(* IEC 61131-3 sources: ml2plc/benchmarks/st (part 14) *)

VAR
    (* Merged variables from all regions *)
    buffer_0 : ARRAY[0..63] OF REAL;
    buffer_1 : ARRAY[0..63] OF REAL;
    c_state_0 : ARRAY[0..63] OF REAL;
    c_state_3 : ARRAY[0..63] OF REAL;
    f_gate_0 : ARRAY[0..63] OF REAL;
    f_gate_3 : ARRAY[0..63] OF REAL;
    g_gate_0 : ARRAY[0..63] OF REAL;
    g_gate_3 : ARRAY[0..63] OF REAL;
    h_state_0 : ARRAY[0..63] OF REAL;
    h_state_3 : ARRAY[0..63] OF REAL;
    i_gate_0 : ARRAY[0..63] OF REAL;
    i_gate_3 : ARRAY[0..63] OF REAL;
    o_gate_0 : ARRAY[0..63] OF REAL;
    o_gate_3 : ARRAY[0..63] OF REAL;

    (* Temporary computation variables *)
    i : DINT;
    j : DINT;
    t : DINT;
    sum : REAL;
    (* Computation helpers *)
    max_val : REAL;
    exp_val : REAL;
    exp_sum : REAL;
    (* Spatial loop variables *)
    oc : DINT;
    oh : DINT;
    ow : DINT;
    ic : DINT;
    kh : DINT;
    kw : DINT;
    ih : DINT;
    iw : DINT;
    (* Transpose loop variables *)
    t2_d0 : DINT;
    t2_d1 : DINT;
    t2_d2 : DINT;
END_VAR

(* Forward pass execution *)

(* Region: r0 [ACYCLIC] *)
(* Acyclic Region r0 *)
(* Layer 0: LSTM (hidden_size=64, input_size=1, seq_len=1) *)
(* Generating output: Y *)

(* Initialize states to zero *)
FOR j := 0 TO 63 DO
    h_state_0[j] := 0.0;
    c_state_0[j] := 0.0;
END_FOR;

(* Process 1 timesteps *)
FOR t := 0 TO 0 DO

    (* Input Gate *)
    FOR j := 0 TO 63 DO
        sum := 0.0;
        FOR i := 0 TO 0 DO
            sum := sum + input_data * weights_0_i[j * 1 + i] ;
        END_FOR;
        FOR i := 0 TO 63 DO
            sum := sum + h_state_0[i] * recurrent_0_i[j * 64 + i] ;
        END_FOR;
    sum := sum + bias_0_i[j];
    i_gate_0[j] := 1.0 / (1.0 + EXP(-sum));
    END_FOR;

    (* Forget Gate *)
    FOR j := 0 TO 63 DO
        sum := 0.0;
        FOR i := 0 TO 0 DO
            sum := sum + input_data * weights_0_f[j * 1 + i] ;
        END_FOR;
        FOR i := 0 TO 63 DO
            sum := sum + h_state_0[i] * recurrent_0_f[j * 64 + i] ;
        END_FOR;
    sum := sum + bias_0_f[j];
    f_gate_0[j] := 1.0 / (1.0 + EXP(-sum));
    END_FOR;

    (* Cell Gate *)
    FOR j := 0 TO 63 DO
        sum := 0.0;
        FOR i := 0 TO 0 DO
            sum := sum + input_data * weights_0_g[j * 1 + i] ;
        END_FOR;
        FOR i := 0 TO 63 DO
            sum := sum + h_state_0[i] * recurrent_0_g[j * 64 + i] ;
        END_FOR;
    sum := sum + bias_0_g[j];
    exp_val := EXP(2.0 * sum);
    g_gate_0[j] := (exp_val - 1.0) / (exp_val + 1.0);
    END_FOR;

    (* Output Gate *)
    FOR j := 0 TO 63 DO
        sum := 0.0;
        FOR i := 0 TO 0 DO
            sum := sum + input_data * weights_0_o[j * 1 + i] ;
        END_FOR;
        FOR i := 0 TO 63 DO
            sum := sum + h_state_0[i] * recurrent_0_o[j * 64 + i] ;
        END_FOR;
    sum := sum + bias_0_o[j];
    o_gate_0[j] := 1.0 / (1.0 + EXP(-sum));
    END_FOR;

    (* Cell state: c_t = f_t * c_{t-1} + i_t * g_t *)
    FOR j := 0 TO 63 DO
        c_state_0[j] := f_gate_0[j] * c_state_0[j] + i_gate_0[j] * g_gate_0[j];
    END_FOR;

    (* Hidden state: h_t = o_t * tanh(c_t) *)
    FOR j := 0 TO 63 DO
        exp_val := EXP(2.0 * c_state_0[j]);
        h_state_0[j] := o_gate_0[j] * ((exp_val - 1.0) / (exp_val + 1.0));
    END_FOR;

    (* Y output: Full sequence *)
    FOR j := 0 TO 63 DO
        buffer_0[t * 64 + j] := h_state_0[j];
    END_FOR;
END_FOR;

(* Layer 1: Squeeze *)
FOR i := 0 TO 63 DO
    buffer_1[i] := buffer_0[i];
END_FOR;

(* Layer 2: Transpose perm=(1, 0, 2)  (1, 1, 64) -> (1, 1, 64) *)
FOR t2_d0 := 0 TO 0 DO
    FOR t2_d1 := 0 TO 0 DO
        FOR t2_d2 := 0 TO 63 DO
            buffer_0[t2_d0 * 64 + t2_d1 * 64 + t2_d2] := buffer_1[t2_d1 * 64 + t2_d0 * 64 + t2_d2];
        END_FOR;
    END_FOR;
END_FOR;

(* Layer 3: LSTM (hidden_size=64, input_size=64, seq_len=1) *)
(* Generating output: Y *)

(* Initialize states to zero *)
FOR j := 0 TO 63 DO
    h_state_3[j] := 0.0;
    c_state_3[j] := 0.0;
END_FOR;

(* Process 1 timesteps *)
FOR t := 0 TO 0 DO

    (* Input Gate *)
    FOR j := 0 TO 63 DO
        sum := 0.0;
        FOR i := 0 TO 63 DO
            sum := sum + buffer_0[t * 64 + i] * weights_3_i[j * 64 + i] ;
        END_FOR;
        FOR i := 0 TO 63 DO
            sum := sum + h_state_3[i] * recurrent_3_i[j * 64 + i] ;
        END_FOR;
    sum := sum + bias_3_i[j];
    i_gate_3[j] := 1.0 / (1.0 + EXP(-sum));
    END_FOR;

    (* Forget Gate *)
    FOR j := 0 TO 63 DO
        sum := 0.0;
        FOR i := 0 TO 63 DO
            sum := sum + buffer_0[t * 64 + i] * weights_3_f[j * 64 + i] ;
        END_FOR;
        FOR i := 0 TO 63 DO
            sum := sum + h_state_3[i] * recurrent_3_f[j * 64 + i] ;
        END_FOR;
    sum := sum + bias_3_f[j];
    f_gate_3[j] := 1.0 / (1.0 + EXP(-sum));
    END_FOR;

    (* Cell Gate *)
    FOR j := 0 TO 63 DO
        sum := 0.0;
        FOR i := 0 TO 63 DO
            sum := sum + buffer_0[t * 64 + i] * weights_3_g[j * 64 + i] ;
        END_FOR;
        FOR i := 0 TO 63 DO
            sum := sum + h_state_3[i] * recurrent_3_g[j * 64 + i] ;
        END_FOR;
    sum := sum + bias_3_g[j];
    exp_val := EXP(2.0 * sum);
    g_gate_3[j] := (exp_val - 1.0) / (exp_val + 1.0);
    END_FOR;

    (* Output Gate *)
    FOR j := 0 TO 63 DO
        sum := 0.0;
        FOR i := 0 TO 63 DO
            sum := sum + buffer_0[t * 64 + i] * weights_3_o[j * 64 + i] ;
        END_FOR;
        FOR i := 0 TO 63 DO
            sum := sum + h_state_3[i] * recurrent_3_o[j * 64 + i] ;
        END_FOR;
    sum := sum + bias_3_o[j];
    o_gate_3[j] := 1.0 / (1.0 + EXP(-sum));
    END_FOR;

    (* Cell state: c_t = f_t * c_{t-1} + i_t * g_t *)
    FOR j := 0 TO 63 DO
        c_state_3[j] := f_gate_3[j] * c_state_3[j] + i_gate_3[j] * g_gate_3[j];
    END_FOR;

    (* Hidden state: h_t = o_t * tanh(c_t) *)
    FOR j := 0 TO 63 DO
        exp_val := EXP(2.0 * c_state_3[j]);
        h_state_3[j] := o_gate_3[j] * ((exp_val - 1.0) / (exp_val + 1.0));
    END_FOR;

    (* Y output: Full sequence *)
    FOR j := 0 TO 63 DO
        buffer_1[t * 64 + j] := h_state_3[j];
    END_FOR;
END_FOR;

(* Layer 4: Squeeze *)
FOR i := 0 TO 63 DO
    buffer_0[i] := buffer_1[i];
END_FOR;

(* Layer 5: Slice starts=[0] ends=[1] axes=[0] steps=[1] *)
FOR i := 0 TO 63 DO
    buffer_1[i] := buffer_0[i];
END_FOR;

(* Layer 6: Squeeze *)
FOR i := 0 TO 63 DO
    buffer_0[i] := buffer_1[i];
END_FOR;

(* Layer 7: Fused Linear + SOFTMAX *)
FOR j := 0 TO 2 DO
    sum := 0.0;
    FOR i := 0 TO 63 DO
        sum := sum + buffer_0[i] * weights_7[i * 3 + j];
    END_FOR;
output_data[j] := sum + bias_7[j];
END_FOR;

(* Softmax: find max *)
max_val := output_data[0];
FOR i := 1 TO 2 DO
    IF output_data[i] > max_val THEN
        max_val := output_data[i];
    END_IF;
END_FOR;

(* Softmax: compute exponentials and sum *)
exp_sum := 0.0;
FOR i := 0 TO 2 DO
    output_data[i] := EXP(output_data[i] - max_val);
    exp_sum := exp_sum + output_data[i];
END_FOR;

(* Softmax: normalize *)
FOR i := 0 TO 2 DO
    output_data[i] := output_data[i] / exp_sum;
END_FOR;

END_FUNCTION_BLOCK

(* ---- MLP1.st ---- *)
FUNCTION_BLOCK MLP1_FB

    (* Model Inputs/Outputs *)
VAR_INPUT
    input_data : REAL;
END_VAR

VAR_OUTPUT
    output_data : ARRAY[0..2] OF REAL;
END_VAR

VAR CONSTANT
    weights_0 : ARRAY[0..7] OF REAL := [-0.39633444, -0.548940063, -0.0548924804, 2.65775609, -0.186861873, 1.99443269, -0.4275029, 2.42555642];
    bias_0 : ARRAY[0..7] OF REAL := [0, 0, 0, -0.386175603, 1.51318884, -0.335069925, 0, -0.41231662];

    weights_1 : ARRAY[0..63] OF REAL := [-0.249718159, 0.355077267, 0.582239211, 0.299669743, 0.560839117, -0.478885651, -0.387439847, 0.0731658936, 0.468102634, 0.0799882412, -0.327028006, 0.219414055, -0.399431229, -0.0365031362, -0.260698169, -0.198557079, -0.294705153, -0.244047046, 0.125463724, 0.588593543, 0.190051973, -0.535617709, -0.0162392259, 0.530301034, 1.90118039, 1.77590561, -0.333346367, -0.0687134862, -0.151702613, -0.455085605, -0.929370284, -1.71230757, 0.0891756192, 0.0794340521, 0.0402879156, -0.0160570145, -0.381342113, -0.337033749, 1.15654266, 1.46721661, 2.8483572, 2.19387126, -0.00236231089, -0.593520105, -0.337822169, -0.402935982, -1.80942917, -2.64788198, -0.0498700142, 0.161640584, -0.224173844, -0.441094339, 0.0303041339, 0.452861011, -0.248058438, -0.0450696349, 2.57059598, 1.8905555, -0.60645926, -0.0833607316, 0.233341992, -0.298924446, -2.09441996, -2.33421278];
    bias_1 : ARRAY[0..7] OF REAL := [-0.133272439, -0.397205234, -0.0605889186, 0, 0, 0, 1.00933897, 1.0929544];

    weights_2 : ARRAY[0..23] OF REAL := [-2.8537457, 0.653815091, 1.25764716, -1.93262327, 0.2645832, 1.83192003, -0.624833703, 0.0545924753, 0.68312341, -0.0164062381, -0.21331352, -0.586643577, -0.673535287, -0.466759026, -0.15310818, -0.313170284, -0.110788405, 0.485940039, 1.39489615, 0.230346501, -2.96772361, 2.38400936, 0.345051408, -2.33157396];
    bias_2 : ARRAY[0..2] OF REAL := [0.0344888456, 0.284831911, -0.563379645];

END_VAR

VAR
    (* Merged variables from all regions *)
    buffer_0 : ARRAY[0..7] OF REAL;
    buffer_1 : ARRAY[0..7] OF REAL;

    (* Temporary computation variables *)
    i : DINT;
    j : DINT;
    t : DINT;
    sum : REAL;
    (* Computation helpers *)
    max_val : REAL;
    exp_val : REAL;
    exp_sum : REAL;
    (* Spatial loop variables *)
    oc : DINT;
    oh : DINT;
    ow : DINT;
    ic : DINT;
    kh : DINT;
    kw : DINT;
    ih : DINT;
    iw : DINT;
END_VAR

(* Forward pass execution *)

(* Region: r0 [ACYCLIC] *)
(* Acyclic Region r0 *)
(* Layer 0: Fused Linear + RELU *)
FOR j := 0 TO 7 DO
    sum := 0.0;
    FOR i := 0 TO 0 DO
        sum := sum + input_data * weights_0[i * 8 + j];
    END_FOR;
buffer_1[j] := MAX(sum + bias_0[j], 0.0);
END_FOR;

(* Layer 1: Fused Linear + RELU *)
FOR j := 0 TO 7 DO
    sum := 0.0;
    FOR i := 0 TO 7 DO
        sum := sum + buffer_1[i] * weights_1[i * 8 + j];
    END_FOR;
buffer_0[j] := MAX(sum + bias_1[j], 0.0);
END_FOR;

(* Layer 2: Fused Linear + SOFTMAX *)
FOR j := 0 TO 2 DO
    sum := 0.0;
    FOR i := 0 TO 7 DO
        sum := sum + buffer_0[i] * weights_2[i * 3 + j];
    END_FOR;
output_data[j] := sum + bias_2[j];
END_FOR;

(* Softmax: find max *)
max_val := output_data[0];
FOR i := 1 TO 2 DO
    IF output_data[i] > max_val THEN
        max_val := output_data[i];
    END_IF;
END_FOR;

(* Softmax: compute exponentials and sum *)
exp_sum := 0.0;
FOR i := 0 TO 2 DO
    output_data[i] := EXP(output_data[i] - max_val);
    exp_sum := exp_sum + output_data[i];
END_FOR;

(* Softmax: normalize *)
FOR i := 0 TO 2 DO
    output_data[i] := output_data[i] / exp_sum;
END_FOR;

END_FUNCTION_BLOCK

(* ---- MLP1_straton.st ---- *)
FUNCTION_BLOCK MLP1_FB

    (* Model Inputs/Outputs *)
VAR_INPUT
    input_data : REAL;
END_VAR

VAR_OUTPUT
    output_data : ARRAY[0..2] OF REAL;
END_VAR

VAR
    CONSTANT weights_0 : ARRAY[0..7] OF REAL := [-0.39633444, -0.548940063, -0.0548924804, 2.65775609, -0.186861873, 1.99443269, -0.4275029, 2.42555642];
    CONSTANT bias_0 : ARRAY[0..7] OF REAL := [0, 0, 0, -0.386175603, 1.51318884, -0.335069925, 0, -0.41231662];
    CONSTANT weights_1 : ARRAY[0..63] OF REAL := [-0.249718159, 0.355077267, 0.582239211, 0.299669743, 0.560839117, -0.478885651, -0.387439847, 0.0731658936, 0.468102634, 0.0799882412, -0.327028006, 0.219414055, -0.399431229, -0.0365031362, -0.260698169, -0.198557079, -0.294705153, -0.244047046, 0.125463724, 0.588593543, 0.190051973, -0.535617709, -0.0162392259, 0.530301034, 1.90118039, 1.77590561, -0.333346367, -0.0687134862, -0.151702613, -0.455085605, -0.929370284, -1.71230757, 0.0891756192, 0.0794340521, 0.0402879156, -0.0160570145, -0.381342113, -0.337033749, 1.15654266, 1.46721661, 2.8483572, 2.19387126, -0.00236231089, -0.593520105, -0.337822169, -0.402935982, -1.80942917, -2.64788198, -0.0498700142, 0.161640584, -0.224173844, -0.441094339, 0.0303041339, 0.452861011, -0.248058438, -0.0450696349, 2.57059598, 1.8905555, -0.60645926, -0.0833607316, 0.233341992, -0.298924446, -2.09441996, -2.33421278];
    CONSTANT bias_1 : ARRAY[0..7] OF REAL := [-0.133272439, -0.397205234, -0.0605889186, 0, 0, 0, 1.00933897, 1.0929544];
    CONSTANT weights_2 : ARRAY[0..23] OF REAL := [-2.8537457, 0.653815091, 1.25764716, -1.93262327, 0.2645832, 1.83192003, -0.624833703, 0.0545924753, 0.68312341, -0.0164062381, -0.21331352, -0.586643577, -0.673535287, -0.466759026, -0.15310818, -0.313170284, -0.110788405, 0.485940039, 1.39489615, 0.230346501, -2.96772361, 2.38400936, 0.345051408, -2.33157396];
    CONSTANT bias_2 : ARRAY[0..2] OF REAL := [0.0344888456, 0.284831911, -0.563379645];
END_VAR

VAR
    (* Merged variables from all regions *)
    buffer_0 : ARRAY[0..7] OF REAL;
    buffer_1 : ARRAY[0..7] OF REAL;

    (* Temporary computation variables *)
    i : DINT;
    j : DINT;
    t : DINT;
    sum : REAL;
    (* Computation helpers *)
    max_val : REAL;
    exp_val : REAL;
    exp_sum : REAL;
    (* Spatial loop variables *)
    oc : DINT;
    oh : DINT;
    ow : DINT;
    ic : DINT;
    kh : DINT;
    kw : DINT;
    ih : DINT;
    iw : DINT;
END_VAR

(* Forward pass execution *)

(* Region: r0 [ACYCLIC] *)
(* Acyclic Region r0 *)
(* Layer 0: Fused Linear + RELU *)
FOR j := 0 TO 7 DO
    sum := 0.0;
    FOR i := 0 TO 0 DO
        sum := sum + input_data * weights_0[i * 8 + j];
    END_FOR;
buffer_1[j] := MAX(sum + bias_0[j], 0.0);
END_FOR;

(* Layer 1: Fused Linear + RELU *)
FOR j := 0 TO 7 DO
    sum := 0.0;
    FOR i := 0 TO 7 DO
        sum := sum + buffer_1[i] * weights_1[i * 8 + j];
    END_FOR;
buffer_0[j] := MAX(sum + bias_1[j], 0.0);
END_FOR;

(* Layer 2: Fused Linear + SOFTMAX *)
FOR j := 0 TO 2 DO
    sum := 0.0;
    FOR i := 0 TO 7 DO
        sum := sum + buffer_0[i] * weights_2[i * 3 + j];
    END_FOR;
output_data[j] := sum + bias_2[j];
END_FOR;

(* Softmax: find max *)
max_val := output_data[0];
FOR i := 1 TO 2 DO
    IF output_data[i] > max_val THEN
        max_val := output_data[i];
    END_IF;
END_FOR;

(* Softmax: compute exponentials and sum *)
exp_sum := 0.0;
FOR i := 0 TO 2 DO
    output_data[i] := EXP(output_data[i] - max_val);
    exp_sum := exp_sum + output_data[i];
END_FOR;

(* Softmax: normalize *)
FOR i := 0 TO 2 DO
    output_data[i] := output_data[i] / exp_sum;
END_FOR;

END_FUNCTION_BLOCK

(* ---- MLP2.st ---- *)
FUNCTION_BLOCK MLP2_FB

    (* Model Inputs/Outputs *)
VAR_INPUT
    input_data : REAL;
END_VAR

VAR_OUTPUT
    output_data : ARRAY[0..2] OF REAL;
END_VAR

VAR CONSTANT
    weights_0 : ARRAY[0..15] OF REAL := [1.43314791, 1.33845091, 0.0506815463, 1.49691188, 1.27512753, 1.58708322, 1.47887564, -0.365204573, -0.308483124, 0.574066639, 1.42833138, 1.61176145, -0.433426589, -0.366151422, -0.0649271607, 1.51271713];
    bias_0 : ARRAY[0..15] OF REAL := [-0.29454121, -0.253037214, -0.0446978658, -0.325126231, -0.236318275, -0.309140831, -0.181606293, 0, 0, 1.27267432, -0.26554206, -0.343669415, 0, 0, 0, -0.280783415];

    weights_1 : ARRAY[0..191] OF REAL := [0.407936037, 1.01749933, -1.20114148, -0.356967181, -1.92732286, 1.20346272, 0.0781332627, 0.110552192, -0.972595394, -0.313477427, -0.218291625, -1.12861526, 0.221315295, 1.45682728, -0.982407808, -0.285307944, -2.18309093, 1.60580647, 0.2185058, 0.064870894, -0.600545108, 0.315021992, -0.448407263, -1.79436421, 0.404721051, -0.0474102646, 0.0530464835, 0.124062717, -0.176960215, -0.155545041, 0.0506753214, -0.437269509, -0.228712574, -0.369052738, -0.429218858, 0.201358885, 0.28686437, 1.53200614, -1.35171425, 0.0549506545, -1.98245513, 1.03874934, -0.184130549, -0.166306764, -1.5724988, -0.127019316, -0.0215409696, -1.40627873, 0.374695808, 0.546456575, -1.01021481, -0.445112586, -1.66891205, 1.26654756, 0.188432008, -0.0941087306, -0.585701585, 0.377527773, -0.314398438, -1.73832321, -0.38970384, 1.36822653, -0.914057195, -0.0957710743, -1.70956862, 1.32042539, -0.0677670836, -0.0267109871, -0.637701869, 0.0480532646, 0.444410801, -0.946867883, -0.393403441, 0.742363334, -0.25676915, -0.0946780145, -0.875564277, 1.52547073, -0.397308588, -0.14911443, -0.00169039122, 0.104037285, 0.213252962, -0.845695674, -0.0459959507, -0.226814017, -0.0849841833, 0.202506483, 0.451363325, -0.283471584, -0.0728154182, 0.458126426, -0.0492827594, -0.389785051, -0.213810101, 0.270405948, -0.295325041, 0.163871646, -0.30711922, 0.163507402, 0.184971035, -0.372719765, -0.345449448, -0.228496328, 0.0936062336, 0.0391324759, 0.284702837, 0.357444406, -0.416430354, -0.491165191, 1.07041216, -0.202913612, 0.692038596, 0.704371512, -0.373513103, -0.401845783, 1.21737754, -0.425899148, -0.141014099, 0.292727947, -0.334978759, 0.967125177, -1.33363903, 0.22960031, -1.47661817, 1.4430207, -0.289626122, -0.17020148, -0.300850689, -0.333540708, -0.419849396, -1.11759806, 0.142602563, 1.46721053, -1.84906495, 0.158245802, -2.41259527, 0.874757349, 0.342971951, -0.173050821, -1.25909066, -0.401011527, -0.45153591, -1.89688873, -0.369080991, -0.308950663, 0.123701572, 0.320791185, 0.127483606, 0.212434173, -0.174650997, 0.416315794, 0.42220372, 0.406279325, -0.151763678, -0.00749960542, 0.278246522, -0.222188339, 0.33904469, -0.0499780774, -0.382376045, 0.301725268, 0.349979341, 0.429802001, 0.243902266, -0.0203652382, -0.207388222, 0.423593044, -0.189736873, 0.163339436, 0.152080178, -0.200317025, 0.307157099, 0.394105434, 0.0754825473, -0.256659746, -0.0376712382, 0.356436849, -0.0464962423, -0.0120930672, 0.1330176, 0.821651697, -1.08929658, 0.0762865543, -1.80090654, 1.69698608, 0.282058746, 0.17900598, -0.978039861, -0.417294323, -0.228806242, -1.15499389];
    bias_1 : ARRAY[0..11] OF REAL := [-0.0375626311, -0.591020405, 0.921454191, 0, 0.725169361, -0.251833826, -0.0172388218, 0, 0.822310686, 0, 0, 0.749954879];

    weights_2 : ARRAY[0..35] OF REAL := [0.597325504, 0.305420995, -0.48944959, -0.391156137, -2.17112041, 2.10054731, 0.8799631, 0.604366958, -2.2579844, 0.277502537, 0.338385344, 0.18559581, 2.05303097, -2.52683377, -1.09150839, -2.28318071, 0.401268154, 1.54289114, 0.420753717, 0.250676453, -0.16422537, -0.26104933, 0.184558988, -0.18064782, 0.678405464, 1.02316344, -1.90771019, 0.412688792, -0.146873921, -0.577244401, 0.539389789, -0.176821679, 0.457258284, 1.71602476, -2.6372664, -1.0096848];
    bias_2 : ARRAY[0..2] OF REAL := [0.00594961783, 0.432862461, -0.599440217];

END_VAR

VAR
    (* Merged variables from all regions *)
    buffer_0 : ARRAY[0..11] OF REAL;
    buffer_1 : ARRAY[0..15] OF REAL;

    (* Temporary computation variables *)
    i : DINT;
    j : DINT;
    t : DINT;
    sum : REAL;
    (* Computation helpers *)
    max_val : REAL;
    exp_val : REAL;
    exp_sum : REAL;
    (* Spatial loop variables *)
    oc : DINT;
    oh : DINT;
    ow : DINT;
    ic : DINT;
    kh : DINT;
    kw : DINT;
    ih : DINT;
    iw : DINT;
END_VAR

(* Forward pass execution *)

(* Region: r0 [ACYCLIC] *)
(* Acyclic Region r0 *)
(* Layer 0: Fused Linear + RELU *)
FOR j := 0 TO 15 DO
    sum := 0.0;
    FOR i := 0 TO 0 DO
        sum := sum + input_data * weights_0[i * 16 + j];
    END_FOR;
buffer_1[j] := MAX(sum + bias_0[j], 0.0);
END_FOR;

(* Layer 1: Fused Linear + RELU *)
FOR j := 0 TO 11 DO
    sum := 0.0;
    FOR i := 0 TO 15 DO
        sum := sum + buffer_1[i] * weights_1[i * 12 + j];
    END_FOR;
buffer_0[j] := MAX(sum + bias_1[j], 0.0);
END_FOR;

(* Layer 2: Fused Linear + SOFTMAX *)
FOR j := 0 TO 2 DO
    sum := 0.0;
    FOR i := 0 TO 11 DO
        sum := sum + buffer_0[i] * weights_2[i * 3 + j];
    END_FOR;
output_data[j] := sum + bias_2[j];
END_FOR;

(* Softmax: find max *)
max_val := output_data[0];
FOR i := 1 TO 2 DO
    IF output_data[i] > max_val THEN
        max_val := output_data[i];
    END_IF;
END_FOR;

(* Softmax: compute exponentials and sum *)
exp_sum := 0.0;
FOR i := 0 TO 2 DO
    output_data[i] := EXP(output_data[i] - max_val);
    exp_sum := exp_sum + output_data[i];
END_FOR;

(* Softmax: normalize *)
FOR i := 0 TO 2 DO
    output_data[i] := output_data[i] / exp_sum;
END_FOR;

END_FUNCTION_BLOCK

(* ---- MLP2_straton.st ---- *)
FUNCTION_BLOCK MLP2_FB

    (* Model Inputs/Outputs *)
VAR_INPUT
    input_data : REAL;
END_VAR

VAR_OUTPUT
    output_data : ARRAY[0..2] OF REAL;
END_VAR

VAR
    CONSTANT weights_0 : ARRAY[0..15] OF REAL := [1.43314791, 1.33845091, 0.0506815463, 1.49691188, 1.27512753, 1.58708322, 1.47887564, -0.365204573, -0.308483124, 0.574066639, 1.42833138, 1.61176145, -0.433426589, -0.366151422, -0.0649271607, 1.51271713];
    CONSTANT bias_0 : ARRAY[0..15] OF REAL := [-0.29454121, -0.253037214, -0.0446978658, -0.325126231, -0.236318275, -0.309140831, -0.181606293, 0, 0, 1.27267432, -0.26554206, -0.343669415, 0, 0, 0, -0.280783415];
    CONSTANT weights_1 : ARRAY[0..191] OF REAL := [0.407936037, 1.01749933, -1.20114148, -0.356967181, -1.92732286, 1.20346272, 0.0781332627, 0.110552192, -0.972595394, -0.313477427, -0.218291625, -1.12861526, 0.221315295, 1.45682728, -0.982407808, -0.285307944, -2.18309093, 1.60580647, 0.2185058, 0.064870894, -0.600545108, 0.315021992, -0.448407263, -1.79436421, 0.404721051, -0.0474102646, 0.0530464835, 0.124062717, -0.176960215, -0.155545041, 0.0506753214, -0.437269509, -0.228712574, -0.369052738, -0.429218858, 0.201358885, 0.28686437, 1.53200614, -1.35171425, 0.0549506545, -1.98245513, 1.03874934, -0.184130549, -0.166306764, -1.5724988, -0.127019316, -0.0215409696, -1.40627873, 0.374695808, 0.546456575, -1.01021481, -0.445112586, -1.66891205, 1.26654756, 0.188432008, -0.0941087306, -0.585701585, 0.377527773, -0.314398438, -1.73832321, -0.38970384, 1.36822653, -0.914057195, -0.0957710743, -1.70956862, 1.32042539, -0.0677670836, -0.0267109871, -0.637701869, 0.0480532646, 0.444410801, -0.946867883, -0.393403441, 0.742363334, -0.25676915, -0.0946780145, -0.875564277, 1.52547073, -0.397308588, -0.14911443, -0.00169039122, 0.104037285, 0.213252962, -0.845695674, -0.0459959507, -0.226814017, -0.0849841833, 0.202506483, 0.451363325, -0.283471584, -0.0728154182, 0.458126426, -0.0492827594, -0.389785051, -0.213810101, 0.270405948, -0.295325041, 0.163871646, -0.30711922, 0.163507402, 0.184971035, -0.372719765, -0.345449448, -0.228496328, 0.0936062336, 0.0391324759, 0.284702837, 0.357444406, -0.416430354, -0.491165191, 1.07041216, -0.202913612, 0.692038596, 0.704371512, -0.373513103, -0.401845783, 1.21737754, -0.425899148, -0.141014099, 0.292727947, -0.334978759, 0.967125177, -1.33363903, 0.22960031, -1.47661817, 1.4430207, -0.289626122, -0.17020148, -0.300850689, -0.333540708, -0.419849396, -1.11759806, 0.142602563, 1.46721053, -1.84906495, 0.158245802, -2.41259527, 0.874757349, 0.342971951, -0.173050821, -1.25909066, -0.401011527, -0.45153591, -1.89688873, -0.369080991, -0.308950663, 0.123701572, 0.320791185, 0.127483606, 0.212434173, -0.174650997, 0.416315794, 0.42220372, 0.406279325, -0.151763678, -0.00749960542, 0.278246522, -0.222188339, 0.33904469, -0.0499780774, -0.382376045, 0.301725268, 0.349979341, 0.429802001, 0.243902266, -0.0203652382, -0.207388222, 0.423593044, -0.189736873, 0.163339436, 0.152080178, -0.200317025, 0.307157099, 0.394105434, 0.0754825473, -0.256659746, -0.0376712382, 0.356436849, -0.0464962423, -0.0120930672, 0.1330176, 0.821651697, -1.08929658, 0.0762865543, -1.80090654, 1.69698608, 0.282058746, 0.17900598, -0.978039861, -0.417294323, -0.228806242, -1.15499389];
    CONSTANT bias_1 : ARRAY[0..11] OF REAL := [-0.0375626311, -0.591020405, 0.921454191, 0, 0.725169361, -0.251833826, -0.0172388218, 0, 0.822310686, 0, 0, 0.749954879];
    CONSTANT weights_2 : ARRAY[0..35] OF REAL := [0.597325504, 0.305420995, -0.48944959, -0.391156137, -2.17112041, 2.10054731, 0.8799631, 0.604366958, -2.2579844, 0.277502537, 0.338385344, 0.18559581, 2.05303097, -2.52683377, -1.09150839, -2.28318071, 0.401268154, 1.54289114, 0.420753717, 0.250676453, -0.16422537, -0.26104933, 0.184558988, -0.18064782, 0.678405464, 1.02316344, -1.90771019, 0.412688792, -0.146873921, -0.577244401, 0.539389789, -0.176821679, 0.457258284, 1.71602476, -2.6372664, -1.0096848];
    CONSTANT bias_2 : ARRAY[0..2] OF REAL := [0.00594961783, 0.432862461, -0.599440217];
END_VAR

VAR
    (* Merged variables from all regions *)
    buffer_0 : ARRAY[0..11] OF REAL;
    buffer_1 : ARRAY[0..15] OF REAL;

    (* Temporary computation variables *)
    i : DINT;
    j : DINT;
    t : DINT;
    sum : REAL;
    (* Computation helpers *)
    max_val : REAL;
    exp_val : REAL;
    exp_sum : REAL;
    (* Spatial loop variables *)
    oc : DINT;
    oh : DINT;
    ow : DINT;
    ic : DINT;
    kh : DINT;
    kw : DINT;
    ih : DINT;
    iw : DINT;
END_VAR

(* Forward pass execution *)

(* Region: r0 [ACYCLIC] *)
(* Acyclic Region r0 *)
(* Layer 0: Fused Linear + RELU *)
FOR j := 0 TO 15 DO
    sum := 0.0;
    FOR i := 0 TO 0 DO
        sum := sum + input_data * weights_0[i * 16 + j];
    END_FOR;
buffer_1[j] := MAX(sum + bias_0[j], 0.0);
END_FOR;

(* Layer 1: Fused Linear + RELU *)
FOR j := 0 TO 11 DO
    sum := 0.0;
    FOR i := 0 TO 15 DO
        sum := sum + buffer_1[i] * weights_1[i * 12 + j];
    END_FOR;
buffer_0[j] := MAX(sum + bias_1[j], 0.0);
END_FOR;

(* Layer 2: Fused Linear + SOFTMAX *)
FOR j := 0 TO 2 DO
    sum := 0.0;
    FOR i := 0 TO 11 DO
        sum := sum + buffer_0[i] * weights_2[i * 3 + j];
    END_FOR;
output_data[j] := sum + bias_2[j];
END_FOR;

(* Softmax: find max *)
max_val := output_data[0];
FOR i := 1 TO 2 DO
    IF output_data[i] > max_val THEN
        max_val := output_data[i];
    END_IF;
END_FOR;

(* Softmax: compute exponentials and sum *)
exp_sum := 0.0;
FOR i := 0 TO 2 DO
    output_data[i] := EXP(output_data[i] - max_val);
    exp_sum := exp_sum + output_data[i];
END_FOR;

(* Softmax: normalize *)
FOR i := 0 TO 2 DO
    output_data[i] := output_data[i] / exp_sum;
END_FOR;

END_FUNCTION_BLOCK

(* ---- MLP3.st ---- *)
FUNCTION_BLOCK MLP3_FB

    (* Model Inputs/Outputs *)
VAR_INPUT
    input_data : REAL;
END_VAR

VAR_OUTPUT
    output_data : ARRAY[0..2] OF REAL;
END_VAR

VAR CONSTANT
    weights_0 : ARRAY[0..15] OF REAL := [-0.00587902591, -0.552422941, 0.967146397, 0.754148066, 1.25726664, 1.11561942, 0.95474416, -0.182324529, 0.328789264, 1.34799659, -0.385122776, -0.0446821451, 0.854335308, -0.216900408, 1.21413243, -0.438498348];
    bias_0 : ARRAY[0..15] OF REAL := [-0.00600522757, 0, -0.189637959, 0.738064468, 0.0427235253, -0.21873486, -0.19639723, 0, 0.694740415, -0.25393635, 0, 0, -0.166762605, 0, -0.225604698, 0];

    weights_1 : ARRAY[0..191] OF REAL := [-0.184632748, 0.405195683, 0.267466664, 0.0684873313, -0.272403359, -0.228539929, 0.0493211746, 0.256188154, -0.0618734173, 0.348178506, -0.0788710117, 0.0386230648, 0.404394388, -0.240164593, 0.284622371, 0.316396415, -0.460191071, 0.175221384, 0.361617148, 0.378937483, 0.281072855, -0.298101962, -0.285237551, -0.103949875, -1.000646, -1.33455193, -0.119448751, 0.663446486, -0.118690312, -0.308231711, 0.196718454, -0.404183537, 1.46282196, 0.320483655, -1.64385271, -1.13940179, 0.509094417, 0.40491423, -0.184621274, 1.01015961, -0.0393494666, -0.269764841, -0.190648049, 0.0307046603, 0.3949534, 0.11252892, 0.329844594, 0.0920630917, -0.41428113, 0.127501324, 0.0815565586, 0.503365874, -0.370055854, -0.204682261, -0.277801275, -0.0172735695, 0.987494528, -0.226065889, -0.0749330893, 0.00975561794, -0.764014304, -1.28692186, -0.136849642, 0.560548484, -0.410659432, 0.127846539, -0.435239673, -0.380198658, 1.07893968, 0.0394562706, -1.54017448, -1.49430203, -0.837658226, -1.3741467, -0.0161108375, 0.714836001, 0.0354768336, 0.184587181, -0.427560806, -0.0522892103, 1.36960292, -0.0954019129, -0.726574898, -1.16550958, -0.156141013, 0.401995003, 0.202450097, 0.147672832, -0.0341677666, -0.268849254, -0.460664004, -0.42492637, -0.16253379, 0.130600929, -0.22815077, -0.126967341, 0.109061316, 0.431140065, -0.221005425, 1.02772689, 0.0376223326, -0.184964627, -0.336410463, 0.0121194208, -0.19831942, -0.322269142, -0.0340373255, 0.634771824, -0.668116391, -1.21975172, 0.216390669, 0.576814353, 0.372669578, 0.190112233, -0.155722409, -0.378851354, 0.871239901, 0.0678931028, -1.41413176, -1.32750046, -0.193424761, -0.453020006, -0.0536833107, 0.240351975, -0.456855804, 0.248503983, 0.0137891769, -0.0663235486, -0.346768439, -0.137402147, -0.308698773, 0.159801126, 0.0471958518, 0.0615314245, 0.256134033, -0.0200264156, -0.184742033, -0.0732097626, 0.0532501936, 0.31175065, -0.118734211, 0.378956795, -0.151903629, 0.0718445182, -0.563162327, -1.0329901, 0.3280918, 0.874449492, -0.0518772602, 0.400076926, 0.444133759, 0.322414011, 1.67673218, 0.0764767304, -1.05872393, -1.33560228, -0.187636614, 0.367284119, 0.382806361, -0.17921257, 0.113314331, 0.434232593, -0.0646075904, 0.391037583, -0.314324051, -0.440758646, 0.334521115, 0.0704363585, -0.766354203, -1.00224555, -0.294651151, 0.515989959, -0.0768560469, -0.27038312, -0.120906442, 0.374218285, 1.33495939, 0.361622036, -1.32872581, -0.784730494, -0.413495719, -0.0494890511, -0.15177238, -0.15318355, -0.413127989, -0.39556551, -0.276276469, -0.381340146, 0.245063305, 0.367093623, 0.0928589702, -0.0233220756];
    bias_1 : ARRAY[0..11] OF REAL := [0.341342688, 0.488520473, 0, 0.56970191, 0, 0, 0, -0.0326530188, -0.33396405, -0.0246085841, 0.299719274, 0.545940161];

    weights_2 : ARRAY[0..95] OF REAL := [-1.81648886, -0.255854517, 1.58292413, 0.224229753, -0.474484146, -0.463809431, -1.10084379, 0.0609974265, -1.31351304, -0.740356982, 1.28859329, 0.321437061, -0.314319193, 0.316025585, -1.43793905, 0.427616745, -0.245407492, -0.485180557, 0.20719099, 0.384393454, 0.394273818, -0.517689466, 0.230686128, 0.264870226, 0.221056968, 0.976806223, 0.732545495, -0.332092792, 0.408505738, -0.0761697739, -0.109968543, -0.274846077, 0.252512336, 0.540791154, -0.015976429, 0.344700575, -0.215772033, -0.131711334, 0.433850765, 0.141305864, 0.129275739, 0.522248626, -0.37742272, 0.49586308, -0.469179839, 0.315679371, -0.228017598, -0.155230999, 0.282684803, 0.0529149771, -0.370359004, 0.262473047, -0.478302658, -0.47957328, 0.399495363, -0.0226950049, -0.335946381, -0.116256997, -0.459948957, -0.292422444, -0.0366530754, -0.404380381, -0.238317788, 0.335635066, 0.916428924, 0.876654625, -1.5151819, -0.217789859, 1.09172642, -0.0582694411, 1.34040082, -0.162317067, -0.0425800346, -0.44222334, 0.154414058, -0.0896951556, 0.142028809, 0.148699135, 0.237090454, 0.51511395, -0.0626033023, -1.84152043, 1.65539598, -0.163748592, -1.54569745, -0.0964944363, 0.701417565, -0.490412295, -1.40768659, -1.1170882, 1.453089, 0.163948908, -0.205052346, -0.224230155, -0.847475111, -0.114188001];
    bias_2 : ARRAY[0..7] OF REAL := [-0.209351003, 0.160942703, 0.502345741, -0.0326822847, 0.17593953, -0.0117381429, -0.12108995, -0.0080464296];

    weights_3 : ARRAY[0..23] OF REAL := [-0.260821044, -1.87934554, 1.76616359, -2.06646132, 1.00641108, 1.05295658, 1.74152339, 0.260352761, -1.73525214, -0.531937897, -0.256840169, 0.124239177, -2.1729877, 1.2575444, 0.0398956165, 0.726067603, 0.445748121, -0.529940963, 0.0432996601, -1.82273531, 1.60026789, -0.593493521, 0.229713753, -0.675501704];
    bias_3 : ARRAY[0..2] OF REAL := [0.0914735422, 0.0294843595, -0.174332708];

END_VAR

VAR
    (* Merged variables from all regions *)
    buffer_0 : ARRAY[0..11] OF REAL;
    buffer_1 : ARRAY[0..15] OF REAL;

    (* Temporary computation variables *)
    i : DINT;
    j : DINT;
    t : DINT;
    sum : REAL;
    (* Computation helpers *)
    max_val : REAL;
    exp_val : REAL;
    exp_sum : REAL;
    (* Spatial loop variables *)
    oc : DINT;
    oh : DINT;
    ow : DINT;
    ic : DINT;
    kh : DINT;
    kw : DINT;
    ih : DINT;
    iw : DINT;
END_VAR

(* Forward pass execution *)

(* Region: r0 [ACYCLIC] *)
(* Acyclic Region r0 *)
(* Layer 0: Fused Linear + RELU *)
FOR j := 0 TO 15 DO
    sum := 0.0;
    FOR i := 0 TO 0 DO
        sum := sum + input_data * weights_0[i * 16 + j];
    END_FOR;
buffer_1[j] := MAX(sum + bias_0[j], 0.0);
END_FOR;

(* Layer 1: Fused Linear + RELU *)
FOR j := 0 TO 11 DO
    sum := 0.0;
    FOR i := 0 TO 15 DO
        sum := sum + buffer_1[i] * weights_1[i * 12 + j];
    END_FOR;
buffer_0[j] := MAX(sum + bias_1[j], 0.0);
END_FOR;

(* Layer 2: Fused Linear + RELU *)
FOR j := 0 TO 7 DO
    sum := 0.0;
    FOR i := 0 TO 11 DO
        sum := sum + buffer_0[i] * weights_2[i * 8 + j];
    END_FOR;
buffer_1[j] := MAX(sum + bias_2[j], 0.0);
END_FOR;

(* Layer 3: Fused Linear + SOFTMAX *)
FOR j := 0 TO 2 DO
    sum := 0.0;
    FOR i := 0 TO 7 DO
        sum := sum + buffer_1[i] * weights_3[i * 3 + j];
    END_FOR;
output_data[j] := sum + bias_3[j];
END_FOR;

(* Softmax: find max *)
max_val := output_data[0];
FOR i := 1 TO 2 DO
    IF output_data[i] > max_val THEN
        max_val := output_data[i];
    END_IF;
END_FOR;

(* Softmax: compute exponentials and sum *)
exp_sum := 0.0;
FOR i := 0 TO 2 DO
    output_data[i] := EXP(output_data[i] - max_val);
    exp_sum := exp_sum + output_data[i];
END_FOR;

(* Softmax: normalize *)
FOR i := 0 TO 2 DO
    output_data[i] := output_data[i] / exp_sum;
END_FOR;

END_FUNCTION_BLOCK

(* ---- MLP3_straton.st ---- *)
FUNCTION_BLOCK MLP3_FB

    (* Model Inputs/Outputs *)
VAR_INPUT
    input_data : REAL;
END_VAR

VAR_OUTPUT
    output_data : ARRAY[0..2] OF REAL;
END_VAR

VAR
    CONSTANT weights_0 : ARRAY[0..15] OF REAL := [-0.00587902591, -0.552422941, 0.967146397, 0.754148066, 1.25726664, 1.11561942, 0.95474416, -0.182324529, 0.328789264, 1.34799659, -0.385122776, -0.0446821451, 0.854335308, -0.216900408, 1.21413243, -0.438498348];
    CONSTANT bias_0 : ARRAY[0..15] OF REAL := [-0.00600522757, 0, -0.189637959, 0.738064468, 0.0427235253, -0.21873486, -0.19639723, 0, 0.694740415, -0.25393635, 0, 0, -0.166762605, 0, -0.225604698, 0];
    CONSTANT weights_1 : ARRAY[0..191] OF REAL := [-0.184632748, 0.405195683, 0.267466664, 0.0684873313, -0.272403359, -0.228539929, 0.0493211746, 0.256188154, -0.0618734173, 0.348178506, -0.0788710117, 0.0386230648, 0.404394388, -0.240164593, 0.284622371, 0.316396415, -0.460191071, 0.175221384, 0.361617148, 0.378937483, 0.281072855, -0.298101962, -0.285237551, -0.103949875, -1.000646, -1.33455193, -0.119448751, 0.663446486, -0.118690312, -0.308231711, 0.196718454, -0.404183537, 1.46282196, 0.320483655, -1.64385271, -1.13940179, 0.509094417, 0.40491423, -0.184621274, 1.01015961, -0.0393494666, -0.269764841, -0.190648049, 0.0307046603, 0.3949534, 0.11252892, 0.329844594, 0.0920630917, -0.41428113, 0.127501324, 0.0815565586, 0.503365874, -0.370055854, -0.204682261, -0.277801275, -0.0172735695, 0.987494528, -0.226065889, -0.0749330893, 0.00975561794, -0.764014304, -1.28692186, -0.136849642, 0.560548484, -0.410659432, 0.127846539, -0.435239673, -0.380198658, 1.07893968, 0.0394562706, -1.54017448, -1.49430203, -0.837658226, -1.3741467, -0.0161108375, 0.714836001, 0.0354768336, 0.184587181, -0.427560806, -0.0522892103, 1.36960292, -0.0954019129, -0.726574898, -1.16550958, -0.156141013, 0.401995003, 0.202450097, 0.147672832, -0.0341677666, -0.268849254, -0.460664004, -0.42492637, -0.16253379, 0.130600929, -0.22815077, -0.126967341, 0.109061316, 0.431140065, -0.221005425, 1.02772689, 0.0376223326, -0.184964627, -0.336410463, 0.0121194208, -0.19831942, -0.322269142, -0.0340373255, 0.634771824, -0.668116391, -1.21975172, 0.216390669, 0.576814353, 0.372669578, 0.190112233, -0.155722409, -0.378851354, 0.871239901, 0.0678931028, -1.41413176, -1.32750046, -0.193424761, -0.453020006, -0.0536833107, 0.240351975, -0.456855804, 0.248503983, 0.0137891769, -0.0663235486, -0.346768439, -0.137402147, -0.308698773, 0.159801126, 0.0471958518, 0.0615314245, 0.256134033, -0.0200264156, -0.184742033, -0.0732097626, 0.0532501936, 0.31175065, -0.118734211, 0.378956795, -0.151903629, 0.0718445182, -0.563162327, -1.0329901, 0.3280918, 0.874449492, -0.0518772602, 0.400076926, 0.444133759, 0.322414011, 1.67673218, 0.0764767304, -1.05872393, -1.33560228, -0.187636614, 0.367284119, 0.382806361, -0.17921257, 0.113314331, 0.434232593, -0.0646075904, 0.391037583, -0.314324051, -0.440758646, 0.334521115, 0.0704363585, -0.766354203, -1.00224555, -0.294651151, 0.515989959, -0.0768560469, -0.27038312, -0.120906442, 0.374218285, 1.33495939, 0.361622036, -1.32872581, -0.784730494, -0.413495719, -0.0494890511, -0.15177238, -0.15318355, -0.413127989, -0.39556551, -0.276276469, -0.381340146, 0.245063305, 0.367093623, 0.0928589702, -0.0233220756];
    CONSTANT bias_1 : ARRAY[0..11] OF REAL := [0.341342688, 0.488520473, 0, 0.56970191, 0, 0, 0, -0.0326530188, -0.33396405, -0.0246085841, 0.299719274, 0.545940161];
    CONSTANT weights_2 : ARRAY[0..95] OF REAL := [-1.81648886, -0.255854517, 1.58292413, 0.224229753, -0.474484146, -0.463809431, -1.10084379, 0.0609974265, -1.31351304, -0.740356982, 1.28859329, 0.321437061, -0.314319193, 0.316025585, -1.43793905, 0.427616745, -0.245407492, -0.485180557, 0.20719099, 0.384393454, 0.394273818, -0.517689466, 0.230686128, 0.264870226, 0.221056968, 0.976806223, 0.732545495, -0.332092792, 0.408505738, -0.0761697739, -0.109968543, -0.274846077, 0.252512336, 0.540791154, -0.015976429, 0.344700575, -0.215772033, -0.131711334, 0.433850765, 0.141305864, 0.129275739, 0.522248626, -0.37742272, 0.49586308, -0.469179839, 0.315679371, -0.228017598, -0.155230999, 0.282684803, 0.0529149771, -0.370359004, 0.262473047, -0.478302658, -0.47957328, 0.399495363, -0.0226950049, -0.335946381, -0.116256997, -0.459948957, -0.292422444, -0.0366530754, -0.404380381, -0.238317788, 0.335635066, 0.916428924, 0.876654625, -1.5151819, -0.217789859, 1.09172642, -0.0582694411, 1.34040082, -0.162317067, -0.0425800346, -0.44222334, 0.154414058, -0.0896951556, 0.142028809, 0.148699135, 0.237090454, 0.51511395, -0.0626033023, -1.84152043, 1.65539598, -0.163748592, -1.54569745, -0.0964944363, 0.701417565, -0.490412295, -1.40768659, -1.1170882, 1.453089, 0.163948908, -0.205052346, -0.224230155, -0.847475111, -0.114188001];
    CONSTANT bias_2 : ARRAY[0..7] OF REAL := [-0.209351003, 0.160942703, 0.502345741, -0.0326822847, 0.17593953, -0.0117381429, -0.12108995, -0.0080464296];
    CONSTANT weights_3 : ARRAY[0..23] OF REAL := [-0.260821044, -1.87934554, 1.76616359, -2.06646132, 1.00641108, 1.05295658, 1.74152339, 0.260352761, -1.73525214, -0.531937897, -0.256840169, 0.124239177, -2.1729877, 1.2575444, 0.0398956165, 0.726067603, 0.445748121, -0.529940963, 0.0432996601, -1.82273531, 1.60026789, -0.593493521, 0.229713753, -0.675501704];
    CONSTANT bias_3 : ARRAY[0..2] OF REAL := [0.0914735422, 0.0294843595, -0.174332708];
END_VAR

VAR
    (* Merged variables from all regions *)
    buffer_0 : ARRAY[0..11] OF REAL;
    buffer_1 : ARRAY[0..15] OF REAL;

    (* Temporary computation variables *)
    i : DINT;
    j : DINT;
    t : DINT;
    sum : REAL;
    (* Computation helpers *)
    max_val : REAL;
    exp_val : REAL;
    exp_sum : REAL;
    (* Spatial loop variables *)
    oc : DINT;
    oh : DINT;
    ow : DINT;
    ic : DINT;
    kh : DINT;
    kw : DINT;
    ih : DINT;
    iw : DINT;
END_VAR

(* Forward pass execution *)

(* Region: r0 [ACYCLIC] *)
(* Acyclic Region r0 *)
(* Layer 0: Fused Linear + RELU *)
FOR j := 0 TO 15 DO
    sum := 0.0;
    FOR i := 0 TO 0 DO
        sum := sum + input_data * weights_0[i * 16 + j];
    END_FOR;
buffer_1[j] := MAX(sum + bias_0[j], 0.0);
END_FOR;

(* Layer 1: Fused Linear + RELU *)
FOR j := 0 TO 11 DO
    sum := 0.0;
    FOR i := 0 TO 15 DO
        sum := sum + buffer_1[i] * weights_1[i * 12 + j];
    END_FOR;
buffer_0[j] := MAX(sum + bias_1[j], 0.0);
END_FOR;

(* Layer 2: Fused Linear + RELU *)
FOR j := 0 TO 7 DO
    sum := 0.0;
    FOR i := 0 TO 11 DO
        sum := sum + buffer_0[i] * weights_2[i * 8 + j];
    END_FOR;
buffer_1[j] := MAX(sum + bias_2[j], 0.0);
END_FOR;

(* Layer 3: Fused Linear + SOFTMAX *)
FOR j := 0 TO 2 DO
    sum := 0.0;
    FOR i := 0 TO 7 DO
        sum := sum + buffer_1[i] * weights_3[i * 3 + j];
    END_FOR;
output_data[j] := sum + bias_3[j];
END_FOR;

(* Softmax: find max *)
max_val := output_data[0];
FOR i := 1 TO 2 DO
    IF output_data[i] > max_val THEN
        max_val := output_data[i];
    END_IF;
END_FOR;

(* Softmax: compute exponentials and sum *)
exp_sum := 0.0;
FOR i := 0 TO 2 DO
    output_data[i] := EXP(output_data[i] - max_val);
    exp_sum := exp_sum + output_data[i];
END_FOR;

(* Softmax: normalize *)
FOR i := 0 TO 2 DO
    output_data[i] := output_data[i] / exp_sum;
END_FOR;

END_FUNCTION_BLOCK

(* ---- MLP4.st ---- *)
FUNCTION_BLOCK MLP4_FB

    (* Model Inputs/Outputs *)
VAR_INPUT
    input_data : REAL;
END_VAR

VAR_OUTPUT
    output_data : ARRAY[0..2] OF REAL;
END_VAR

VAR CONSTANT
    weights_0 : ARRAY[0..11] OF REAL := [-0.000433303358, -0.259365618, -0.391792595, 0.892193496, -0.21629557, 0.906598866, 0.674373746, -0.558652401, 0.797402382, -0.203392595, -0.0916015506, -0.275554031];
    bias_0 : ARRAY[0..11] OF REAL := [-0.01485065, 0, 0, -0.110643201, 0, -0.10883344, 0.494125873, 0, -0.0718084425, 0, 0, 0.0934562832];

    weights_1 : ARRAY[0..143] OF REAL := [-0.298880816, -0.00152957439, 0.474849463, 0.306986213, -0.405141115, 0.48761344, 0.102969885, -0.344942093, -0.025667632, 0.300008178, 0.0242930651, 0.0812352896, -0.399855614, 0.342774987, -0.167612314, -0.202104092, 0.400625467, 0.0856477022, -0.28502667, 0.138476968, -0.497452259, 0.148318172, 0.0338615179, 0.0765039921, 0.455938458, 0.437605858, -0.0340754986, 0.0788701773, 0.216484904, -0.378376842, 0.0994442701, 0.21826601, 0.0169439316, 0.127574921, 0.0280764103, -0.241563201, 0.466122746, -0.699138701, -0.465045094, 0.169780999, 0.0941107273, -0.805239379, 0.0534801483, -0.662550032, -0.685605705, 0.968525112, -0.460680127, -0.166365623, 0.0986363888, 0.0149536133, 0.134114027, 0.112850904, -0.322958112, 0.000517606735, 0.00420176983, -0.265694261, 0.0301915407, -0.36379385, 0.25820291, 0.235822558, -0.345233202, -0.653570831, 0.385483146, -0.00680492818, -0.49095428, -0.515505373, -0.114819884, -0.382326335, -0.359407783, 0.961687744, -0.338742614, 0.0313850641, -0.435787201, 0.347338021, -0.214350343, 0.761085331, -0.226865888, 0.161012426, -0.0433943272, 0.119208843, 0.336905152, 0.277065068, -0.440087557, -0.233440638, 0.408263087, -0.104699612, -0.361725569, 0.311339378, -0.227642298, 0.0617007017, -0.293772459, 0.384199858, 0.164174676, 0.414742708, 0.433134317, -0.404003978, 0.182819128, -0.330298752, -0.125009775, 0.285753429, -0.197088599, -0.408124834, -0.472592235, 0.0365833901, -0.511666477, 0.983981192, 0.0605376959, -0.0932275057, -0.190840483, -0.154848933, -0.0741977692, -0.151085258, 0.326916337, 0.134229302, 0.337689042, 0.491287947, -0.43740499, 0.129448891, 0.0393525362, 0.239477754, 0.19716692, -0.477047086, 0.177004576, 0.481723666, 0.269957662, 0.416185498, 0.459372401, -0.413143158, -0.338309169, -0.127821088, -0.000163674355, 0.21434617, 0.0654553175, 0.275052726, 0.232549548, 0.462537229, -0.277248025, 0.566420615, -0.0154316425, 0.0670012161, 0.322845042, -0.703867555, -0.42449069, 0.0752505064];
    bias_1 : ARRAY[0..11] OF REAL := [0, 0.0762805939, 0, 0.427145034, 0, 0.265131414, 0, 0.104791395, 0.163058564, -0.0698945299, 0, 0];

    weights_2 : ARRAY[0..143] OF REAL := [-0.0732795, -0.0192222595, -0.0223456621, 0.238418102, 0.42742753, 0.387707472, 0.0560674667, 0.497440934, -0.188100457, 0.140284061, 0.00321984291, 0.216849923, 0.713741481, 1.14185643, 0.364514828, -0.272081375, 0.298052073, 0.77692169, 0.136832684, -0.306305498, -0.110322058, 0.666837156, -0.950240552, -0.577573478, -0.0160051584, 0.136987567, -0.139540672, 0.423784018, -0.0908498764, 0.0130108595, -0.378936529, 0.397712588, 0.061617136, 0.433579922, 0.0201644897, -0.362152457, 0.269566983, 0.333628774, -0.199544549, -0.256773472, -0.191290855, 0.425239295, 0.431172222, 0.422367722, -0.00804625079, 0.283771634, 0.738150299, -0.0722901151, 0.345920205, -0.16432035, -0.190850139, 0.153236985, 0.41677928, 0.191761374, 0.0371178389, -0.150701284, -0.228767514, -0.487576485, -0.431827307, 0.115035653, 0.662138462, 0.310151964, -0.236443281, -0.365703464, 0.177370906, 0.856746972, 0.852512956, -0.452390254, -0.177463084, 0.976620197, -0.163254559, -0.203274101, 0.0719256401, -0.0631088018, 0.406458139, 0.0234757662, 0.462169051, -0.442534924, 0.354242206, -0.44355011, -0.0484654903, 0.226473331, 0.212472558, 0.420234323, 0.426062226, 0.848032057, 0.128262877, -0.346981406, 0.291216612, 0.198882177, 0.931373537, -0.17434077, -0.829320014, 0.596504033, -0.494588077, -0.319661349, 0.52673316, 0.658886313, -0.390596747, 0.164096832, -0.349671721, 0.827856123, 0.214752108, -0.386913747, -0.563117087, 0.336437672, -0.081583716, -0.159346983, -0.834958732, 0.257420421, -0.184664369, -0.0109804869, 0.000288844109, -0.102150165, -0.867207229, 0.92633605, 0.984464109, -0.707509458, 1.02899325, 0.851662636, 0.354382038, -0.145519614, 0.169264793, -0.401280165, -0.128762484, -0.172792196, -0.218239188, -0.0484528542, -0.459516287, 0.0344768763, 0.407926202, 0.413538814, -0.200879812, -0.290590405, 0.373239398, 0.0639884472, 0.32487762, 0.184734344, -0.0577995777, 0.486539602, 0.13507998, -0.303152323, 0.348408341, 0.190643311];
    bias_2 : ARRAY[0..11] OF REAL := [0.268908471, 0.419366419, 0, 0, 0, 0.313713729, 0.197716802, -0.0247089025, -0.00207538903, 0.286986262, 0.198602244, -0.0521202013];

    weights_3 : ARRAY[0..143] OF REAL := [-0.357495427, -0.307849735, -0.416388512, -0.0850503445, -0.448468804, 1.07230294, 0.370020866, -0.299492478, -0.722271144, -0.303815573, -0.366407573, 0.986412048, -0.22380197, 0.411702961, -0.494180143, -0.191248655, -0.520082176, 0.523566544, -0.239420772, 0.0257567279, 0.0666296035, -0.362573922, 0.534610689, 0.773202121, 0.276561499, 0.0454052687, 0.0226814747, 0.499738216, 0.0659197569, 0.489770055, 0.332119465, 0.490028977, -0.194036484, -0.299536347, 0.358960152, -0.238898873, 0.123157024, 0.0393670797, 0.180379391, 0.470559955, 0.233510375, -0.133527875, -0.272634625, 0.30077076, 0.356262326, -0.332687855, -0.404446244, 0.417606473, 0.0290625095, -0.220114231, -0.200132966, 0.164584398, -0.129657626, -0.309647918, -0.124839902, 0.0649834871, 0.154951215, 0.12078023, -0.198447108, -0.338992834, -0.384413242, -0.0676555261, 0.243490413, -0.0224215984, 0.419704884, 0.399650902, 0.175193667, -0.388169378, 0.205466524, 0.164588884, 0.119603366, 0.904532671, 0.0230317116, -0.80870527, 0.289435983, 0.0350148678, -0.016607346, 0.444647133, 0.0242673159, 0.229468584, -0.732327104, -0.841991127, -0.325898319, 1.03079927, -0.12533319, 0.696952283, -0.137089863, -0.418627381, -0.229799584, -0.760831952, -0.0515791178, 0.0489806756, 0.849764764, -0.0538823716, 0.926742852, -0.362278908, 0.163343668, 1.14239967, 0.269085795, 0.311249375, -0.1962955, -0.426426888, -0.337019682, 0.0170502663, 0.873662829, 0.192067161, 0.693036854, -1.00146031, -0.447796464, -0.385757178, -0.231265187, -0.106191754, 0.171909496, 0.809488177, -0.397168875, -0.263619542, 0.0511783883, -0.836772621, -0.727877676, 1.17547035, -0.103365898, 0.831905544, -0.217022225, -0.419677734, 0.15053536, 0.0626083016, -0.203929305, -0.0176051632, 0.713163078, 0.491280258, 1.0963397, -0.0843987241, -0.496840119, 0.620099068, 0.354867846, -0.366894484, -0.206087083, -1.13332653, -0.214713931, -0.256117702, 0.921475649, 0.3023718, 0.913246453, -1.10309541];
    bias_3 : ARRAY[0..11] OF REAL := [0, 0.119710997, -0.00997092109, 0, -0.00180400128, 0.243082359, 0, -0.00515343109, 0.145769224, -0.137557253, 0.350063741, 0.312690645];

    weights_4 : ARRAY[0..143] OF REAL := [0.450706244, -0.341911197, -0.454755664, -0.063834548, -0.357831359, -0.276776195, 0.301605582, 0.495445967, 0.303405285, -0.30096972, -0.376701355, -0.130076766, -0.300299644, -0.430371284, -0.51883167, -0.84268868, -0.287088871, -0.109367259, -0.817286849, 0.909729838, -0.364345223, -0.380807519, 0.161143929, 0.100938745, 0.0374554396, 0.218073368, -0.281522155, -0.174941421, -0.37441051, 0.0506789684, 0.0436292887, -0.0927791074, 0.47244668, -0.36142385, 0.327807456, 0.472998738, 0.190690041, 0.213500023, 0.425210118, -0.213574409, 0.163247466, 0.419484854, -0.218418241, -0.112340212, -0.400529623, 0.443802476, 0.357275009, -0.401218772, -0.0335019007, -0.125037313, -0.185095012, 0.170340389, -0.201058984, -0.455673128, 0.217301518, -0.38702932, 0.214139879, 0.431893885, 0.488917947, -0.439485908, -0.19993034, 0.322346568, 1.14306962, 0.749802947, -0.373077631, 0.804487646, 0.77006501, -0.550892115, -0.0832547173, -0.298211604, -0.332630187, 0.805645168, 0.368081808, -0.360151887, 0.435218573, 0.324298859, -0.196251392, -0.455414176, 0.147471786, -0.365893245, -0.250006795, 0.143167973, -0.493285775, -0.0164135695, 0.127878308, -0.357789874, -0.443840533, -0.342483342, 0.218469262, 0.170943871, -0.0552097447, 0.0616960526, 0.153929442, 0.374329329, 0.381393313, -0.305997193, 0.36288327, -0.135337353, 0.0422162116, -0.927169621, 0.0343397856, -0.211289778, -0.844623089, 0.929481864, -0.0883726105, 0.199234247, 0.331276417, -0.101934858, 0.401151687, 0.248295903, -0.302112967, -0.459259838, -0.15229702, -1.80295289, 0.310522586, 0.80208832, 0.0157887768, -0.396735907, -0.276871234, -1.69113529, -0.143170267, 0.0102803707, 0.14509201, -0.476439834, 0.204934001, 0.294055164, -0.629547834, 0.928040624, -0.351497144, -0.26870656, -0.409520328, 0.00686698314, -0.354189754, -0.278342724, 0.83324641, 0.794706464, -0.455154419, 1.22785282, 0.826641798, -0.369872659, 0.0869283378, -0.0698348582, -0.122125052, 1.26005256];
    bias_4 : ARRAY[0..11] OF REAL := [-0.0211661961, 0, 0.261660874, -0.0140484339, 0, 0.364149809, 0.144630164, 0.339143276, -0.0598276779, -0.00512596732, -0.0318891779, 0.40167141];

    weights_5 : ARRAY[0..35] OF REAL := [0.173672497, 0.297189862, 0.192978173, 0.289213598, 0.37582773, 0.30365479, 0.627732277, 0.429832458, -1.44617391, 1.52943027, -1.05059588, -0.00112121843, -0.252201021, 0.505529344, -0.516346693, -0.213808402, 0.146612033, -1.31478655, 1.03269589, -0.734977663, -0.726943493, -0.880188823, 0.478668094, 1.19996989, -0.309403777, -0.0974165127, 0.0823692605, -0.150946915, -0.494235575, 0.57968545, 0.0338293761, -0.20537369, -0.302375942, 0.441371918, 0.83744365, -0.748067141];
    bias_5 : ARRAY[0..2] OF REAL := [-0.2327815, 0.190008208, 0.0320904478];

END_VAR

VAR
    (* Merged variables from all regions *)
    buffer_0 : ARRAY[0..11] OF REAL;
    buffer_1 : ARRAY[0..11] OF REAL;

    (* Temporary computation variables *)
    i : DINT;
    j : DINT;
    t : DINT;
    sum : REAL;
    (* Computation helpers *)
    max_val : REAL;
    exp_val : REAL;
    exp_sum : REAL;
    (* Spatial loop variables *)
    oc : DINT;
    oh : DINT;
    ow : DINT;
    ic : DINT;
    kh : DINT;
    kw : DINT;
    ih : DINT;
    iw : DINT;
END_VAR

(* Forward pass execution *)

(* Region: r0 [ACYCLIC] *)
(* Acyclic Region r0 *)
(* Layer 0: Fused Linear + RELU *)
FOR j := 0 TO 11 DO
    sum := 0.0;
    FOR i := 0 TO 0 DO
        sum := sum + input_data * weights_0[i * 12 + j];
    END_FOR;
buffer_1[j] := MAX(sum + bias_0[j], 0.0);
END_FOR;

(* Layer 1: Fused Linear + RELU *)
FOR j := 0 TO 11 DO
    sum := 0.0;
    FOR i := 0 TO 11 DO
        sum := sum + buffer_1[i] * weights_1[i * 12 + j];
    END_FOR;
buffer_0[j] := MAX(sum + bias_1[j], 0.0);
END_FOR;

(* Layer 2: Fused Linear + RELU *)
FOR j := 0 TO 11 DO
    sum := 0.0;
    FOR i := 0 TO 11 DO
        sum := sum + buffer_0[i] * weights_2[i * 12 + j];
    END_FOR;
buffer_1[j] := MAX(sum + bias_2[j], 0.0);
END_FOR;

(* Layer 3: Fused Linear + RELU *)
FOR j := 0 TO 11 DO
    sum := 0.0;
    FOR i := 0 TO 11 DO
        sum := sum + buffer_1[i] * weights_3[i * 12 + j];
    END_FOR;
buffer_0[j] := MAX(sum + bias_3[j], 0.0);
END_FOR;

(* Layer 4: Fused Linear + RELU *)
FOR j := 0 TO 11 DO
    sum := 0.0;
    FOR i := 0 TO 11 DO
        sum := sum + buffer_0[i] * weights_4[i * 12 + j];
    END_FOR;
buffer_1[j] := MAX(sum + bias_4[j], 0.0);
END_FOR;

(* Layer 5: Fused Linear + SOFTMAX *)
FOR j := 0 TO 2 DO
    sum := 0.0;
    FOR i := 0 TO 11 DO
        sum := sum + buffer_1[i] * weights_5[i * 3 + j];
    END_FOR;
output_data[j] := sum + bias_5[j];
END_FOR;

(* Softmax: find max *)
max_val := output_data[0];
FOR i := 1 TO 2 DO
    IF output_data[i] > max_val THEN
        max_val := output_data[i];
    END_IF;
END_FOR;

(* Softmax: compute exponentials and sum *)
exp_sum := 0.0;
FOR i := 0 TO 2 DO
    output_data[i] := EXP(output_data[i] - max_val);
    exp_sum := exp_sum + output_data[i];
END_FOR;

(* Softmax: normalize *)
FOR i := 0 TO 2 DO
    output_data[i] := output_data[i] / exp_sum;
END_FOR;

END_FUNCTION_BLOCK

(* ---- MLP4_straton.st ---- *)
FUNCTION_BLOCK MLP4_FB

    (* Model Inputs/Outputs *)
VAR_INPUT
    input_data : REAL;
END_VAR

VAR_OUTPUT
    output_data : ARRAY[0..2] OF REAL;
END_VAR

VAR
    CONSTANT weights_0 : ARRAY[0..11] OF REAL := [-0.000433303358, -0.259365618, -0.391792595, 0.892193496, -0.21629557, 0.906598866, 0.674373746, -0.558652401, 0.797402382, -0.203392595, -0.0916015506, -0.275554031];
    CONSTANT bias_0 : ARRAY[0..11] OF REAL := [-0.01485065, 0, 0, -0.110643201, 0, -0.10883344, 0.494125873, 0, -0.0718084425, 0, 0, 0.0934562832];
    CONSTANT weights_1 : ARRAY[0..143] OF REAL := [-0.298880816, -0.00152957439, 0.474849463, 0.306986213, -0.405141115, 0.48761344, 0.102969885, -0.344942093, -0.025667632, 0.300008178, 0.0242930651, 0.0812352896, -0.399855614, 0.342774987, -0.167612314, -0.202104092, 0.400625467, 0.0856477022, -0.28502667, 0.138476968, -0.497452259, 0.148318172, 0.0338615179, 0.0765039921, 0.455938458, 0.437605858, -0.0340754986, 0.0788701773, 0.216484904, -0.378376842, 0.0994442701, 0.21826601, 0.0169439316, 0.127574921, 0.0280764103, -0.241563201, 0.466122746, -0.699138701, -0.465045094, 0.169780999, 0.0941107273, -0.805239379, 0.0534801483, -0.662550032, -0.685605705, 0.968525112, -0.460680127, -0.166365623, 0.0986363888, 0.0149536133, 0.134114027, 0.112850904, -0.322958112, 0.000517606735, 0.00420176983, -0.265694261, 0.0301915407, -0.36379385, 0.25820291, 0.235822558, -0.345233202, -0.653570831, 0.385483146, -0.00680492818, -0.49095428, -0.515505373, -0.114819884, -0.382326335, -0.359407783, 0.961687744, -0.338742614, 0.0313850641, -0.435787201, 0.347338021, -0.214350343, 0.761085331, -0.226865888, 0.161012426, -0.0433943272, 0.119208843, 0.336905152, 0.277065068, -0.440087557, -0.233440638, 0.408263087, -0.104699612, -0.361725569, 0.311339378, -0.227642298, 0.0617007017, -0.293772459, 0.384199858, 0.164174676, 0.414742708, 0.433134317, -0.404003978, 0.182819128, -0.330298752, -0.125009775, 0.285753429, -0.197088599, -0.408124834, -0.472592235, 0.0365833901, -0.511666477, 0.983981192, 0.0605376959, -0.0932275057, -0.190840483, -0.154848933, -0.0741977692, -0.151085258, 0.326916337, 0.134229302, 0.337689042, 0.491287947, -0.43740499, 0.129448891, 0.0393525362, 0.239477754, 0.19716692, -0.477047086, 0.177004576, 0.481723666, 0.269957662, 0.416185498, 0.459372401, -0.413143158, -0.338309169, -0.127821088, -0.000163674355, 0.21434617, 0.0654553175, 0.275052726, 0.232549548, 0.462537229, -0.277248025, 0.566420615, -0.0154316425, 0.0670012161, 0.322845042, -0.703867555, -0.42449069, 0.0752505064];
    CONSTANT bias_1 : ARRAY[0..11] OF REAL := [0, 0.0762805939, 0, 0.427145034, 0, 0.265131414, 0, 0.104791395, 0.163058564, -0.0698945299, 0, 0];
    CONSTANT weights_2 : ARRAY[0..143] OF REAL := [-0.0732795, -0.0192222595, -0.0223456621, 0.238418102, 0.42742753, 0.387707472, 0.0560674667, 0.497440934, -0.188100457, 0.140284061, 0.00321984291, 0.216849923, 0.713741481, 1.14185643, 0.364514828, -0.272081375, 0.298052073, 0.77692169, 0.136832684, -0.306305498, -0.110322058, 0.666837156, -0.950240552, -0.577573478, -0.0160051584, 0.136987567, -0.139540672, 0.423784018, -0.0908498764, 0.0130108595, -0.378936529, 0.397712588, 0.061617136, 0.433579922, 0.0201644897, -0.362152457, 0.269566983, 0.333628774, -0.199544549, -0.256773472, -0.191290855, 0.425239295, 0.431172222, 0.422367722, -0.00804625079, 0.283771634, 0.738150299, -0.0722901151, 0.345920205, -0.16432035, -0.190850139, 0.153236985, 0.41677928, 0.191761374, 0.0371178389, -0.150701284, -0.228767514, -0.487576485, -0.431827307, 0.115035653, 0.662138462, 0.310151964, -0.236443281, -0.365703464, 0.177370906, 0.856746972, 0.852512956, -0.452390254, -0.177463084, 0.976620197, -0.163254559, -0.203274101, 0.0719256401, -0.0631088018, 0.406458139, 0.0234757662, 0.462169051, -0.442534924, 0.354242206, -0.44355011, -0.0484654903, 0.226473331, 0.212472558, 0.420234323, 0.426062226, 0.848032057, 0.128262877, -0.346981406, 0.291216612, 0.198882177, 0.931373537, -0.17434077, -0.829320014, 0.596504033, -0.494588077, -0.319661349, 0.52673316, 0.658886313, -0.390596747, 0.164096832, -0.349671721, 0.827856123, 0.214752108, -0.386913747, -0.563117087, 0.336437672, -0.081583716, -0.159346983, -0.834958732, 0.257420421, -0.184664369, -0.0109804869, 0.000288844109, -0.102150165, -0.867207229, 0.92633605, 0.984464109, -0.707509458, 1.02899325, 0.851662636, 0.354382038, -0.145519614, 0.169264793, -0.401280165, -0.128762484, -0.172792196, -0.218239188, -0.0484528542, -0.459516287, 0.0344768763, 0.407926202, 0.413538814, -0.200879812, -0.290590405, 0.373239398, 0.0639884472, 0.32487762, 0.184734344, -0.0577995777, 0.486539602, 0.13507998, -0.303152323, 0.348408341, 0.190643311];
    CONSTANT bias_2 : ARRAY[0..11] OF REAL := [0.268908471, 0.419366419, 0, 0, 0, 0.313713729, 0.197716802, -0.0247089025, -0.00207538903, 0.286986262, 0.198602244, -0.0521202013];
    CONSTANT weights_3 : ARRAY[0..143] OF REAL := [-0.357495427, -0.307849735, -0.416388512, -0.0850503445, -0.448468804, 1.07230294, 0.370020866, -0.299492478, -0.722271144, -0.303815573, -0.366407573, 0.986412048, -0.22380197, 0.411702961, -0.494180143, -0.191248655, -0.520082176, 0.523566544, -0.239420772, 0.0257567279, 0.0666296035, -0.362573922, 0.534610689, 0.773202121, 0.276561499, 0.0454052687, 0.0226814747, 0.499738216, 0.0659197569, 0.489770055, 0.332119465, 0.490028977, -0.194036484, -0.299536347, 0.358960152, -0.238898873, 0.123157024, 0.0393670797, 0.180379391, 0.470559955, 0.233510375, -0.133527875, -0.272634625, 0.30077076, 0.356262326, -0.332687855, -0.404446244, 0.417606473, 0.0290625095, -0.220114231, -0.200132966, 0.164584398, -0.129657626, -0.309647918, -0.124839902, 0.0649834871, 0.154951215, 0.12078023, -0.198447108, -0.338992834, -0.384413242, -0.0676555261, 0.243490413, -0.0224215984, 0.419704884, 0.399650902, 0.175193667, -0.388169378, 0.205466524, 0.164588884, 0.119603366, 0.904532671, 0.0230317116, -0.80870527, 0.289435983, 0.0350148678, -0.016607346, 0.444647133, 0.0242673159, 0.229468584, -0.732327104, -0.841991127, -0.325898319, 1.03079927, -0.12533319, 0.696952283, -0.137089863, -0.418627381, -0.229799584, -0.760831952, -0.0515791178, 0.0489806756, 0.849764764, -0.0538823716, 0.926742852, -0.362278908, 0.163343668, 1.14239967, 0.269085795, 0.311249375, -0.1962955, -0.426426888, -0.337019682, 0.0170502663, 0.873662829, 0.192067161, 0.693036854, -1.00146031, -0.447796464, -0.385757178, -0.231265187, -0.106191754, 0.171909496, 0.809488177, -0.397168875, -0.263619542, 0.0511783883, -0.836772621, -0.727877676, 1.17547035, -0.103365898, 0.831905544, -0.217022225, -0.419677734, 0.15053536, 0.0626083016, -0.203929305, -0.0176051632, 0.713163078, 0.491280258, 1.0963397, -0.0843987241, -0.496840119, 0.620099068, 0.354867846, -0.366894484, -0.206087083, -1.13332653, -0.214713931, -0.256117702, 0.921475649, 0.3023718, 0.913246453, -1.10309541];
    CONSTANT bias_3 : ARRAY[0..11] OF REAL := [0, 0.119710997, -0.00997092109, 0, -0.00180400128, 0.243082359, 0, -0.00515343109, 0.145769224, -0.137557253, 0.350063741, 0.312690645];
    CONSTANT weights_4 : ARRAY[0..143] OF REAL := [0.450706244, -0.341911197, -0.454755664, -0.063834548, -0.357831359, -0.276776195, 0.301605582, 0.495445967, 0.303405285, -0.30096972, -0.376701355, -0.130076766, -0.300299644, -0.430371284, -0.51883167, -0.84268868, -0.287088871, -0.109367259, -0.817286849, 0.909729838, -0.364345223, -0.380807519, 0.161143929, 0.100938745, 0.0374554396, 0.218073368, -0.281522155, -0.174941421, -0.37441051, 0.0506789684, 0.0436292887, -0.0927791074, 0.47244668, -0.36142385, 0.327807456, 0.472998738, 0.190690041, 0.213500023, 0.425210118, -0.213574409, 0.163247466, 0.419484854, -0.218418241, -0.112340212, -0.400529623, 0.443802476, 0.357275009, -0.401218772, -0.0335019007, -0.125037313, -0.185095012, 0.170340389, -0.201058984, -0.455673128, 0.217301518, -0.38702932, 0.214139879, 0.431893885, 0.488917947, -0.439485908, -0.19993034, 0.322346568, 1.14306962, 0.749802947, -0.373077631, 0.804487646, 0.77006501, -0.550892115, -0.0832547173, -0.298211604, -0.332630187, 0.805645168, 0.368081808, -0.360151887, 0.435218573, 0.324298859, -0.196251392, -0.455414176, 0.147471786, -0.365893245, -0.250006795, 0.143167973, -0.493285775, -0.0164135695, 0.127878308, -0.357789874, -0.443840533, -0.342483342, 0.218469262, 0.170943871, -0.0552097447, 0.0616960526, 0.153929442, 0.374329329, 0.381393313, -0.305997193, 0.36288327, -0.135337353, 0.0422162116, -0.927169621, 0.0343397856, -0.211289778, -0.844623089, 0.929481864, -0.0883726105, 0.199234247, 0.331276417, -0.101934858, 0.401151687, 0.248295903, -0.302112967, -0.459259838, -0.15229702, -1.80295289, 0.310522586, 0.80208832, 0.0157887768, -0.396735907, -0.276871234, -1.69113529, -0.143170267, 0.0102803707, 0.14509201, -0.476439834, 0.204934001, 0.294055164, -0.629547834, 0.928040624, -0.351497144, -0.26870656, -0.409520328, 0.00686698314, -0.354189754, -0.278342724, 0.83324641, 0.794706464, -0.455154419, 1.22785282, 0.826641798, -0.369872659, 0.0869283378, -0.0698348582, -0.122125052, 1.26005256];
    CONSTANT bias_4 : ARRAY[0..11] OF REAL := [-0.0211661961, 0, 0.261660874, -0.0140484339, 0, 0.364149809, 0.144630164, 0.339143276, -0.0598276779, -0.00512596732, -0.0318891779, 0.40167141];
    CONSTANT weights_5 : ARRAY[0..35] OF REAL := [0.173672497, 0.297189862, 0.192978173, 0.289213598, 0.37582773, 0.30365479, 0.627732277, 0.429832458, -1.44617391, 1.52943027, -1.05059588, -0.00112121843, -0.252201021, 0.505529344, -0.516346693, -0.213808402, 0.146612033, -1.31478655, 1.03269589, -0.734977663, -0.726943493, -0.880188823, 0.478668094, 1.19996989, -0.309403777, -0.0974165127, 0.0823692605, -0.150946915, -0.494235575, 0.57968545, 0.0338293761, -0.20537369, -0.302375942, 0.441371918, 0.83744365, -0.748067141];
    CONSTANT bias_5 : ARRAY[0..2] OF REAL := [-0.2327815, 0.190008208, 0.0320904478];
END_VAR

VAR
    (* Merged variables from all regions *)
    buffer_0 : ARRAY[0..11] OF REAL;
    buffer_1 : ARRAY[0..11] OF REAL;

    (* Temporary computation variables *)
    i : DINT;
    j : DINT;
    t : DINT;
    sum : REAL;
    (* Computation helpers *)
    max_val : REAL;
    exp_val : REAL;
    exp_sum : REAL;
    (* Spatial loop variables *)
    oc : DINT;
    oh : DINT;
    ow : DINT;
    ic : DINT;
    kh : DINT;
    kw : DINT;
    ih : DINT;
    iw : DINT;
END_VAR

(* Forward pass execution *)

(* Region: r0 [ACYCLIC] *)
(* Acyclic Region r0 *)
(* Layer 0: Fused Linear + RELU *)
FOR j := 0 TO 11 DO
    sum := 0.0;
    FOR i := 0 TO 0 DO
        sum := sum + input_data * weights_0[i * 12 + j];
    END_FOR;
buffer_1[j] := MAX(sum + bias_0[j], 0.0);
END_FOR;

(* Layer 1: Fused Linear + RELU *)
FOR j := 0 TO 11 DO
    sum := 0.0;
    FOR i := 0 TO 11 DO
        sum := sum + buffer_1[i] * weights_1[i * 12 + j];
    END_FOR;
buffer_0[j] := MAX(sum + bias_1[j], 0.0);
END_FOR;

(* Layer 2: Fused Linear + RELU *)
FOR j := 0 TO 11 DO
    sum := 0.0;
    FOR i := 0 TO 11 DO
        sum := sum + buffer_0[i] * weights_2[i * 12 + j];
    END_FOR;
buffer_1[j] := MAX(sum + bias_2[j], 0.0);
END_FOR;

(* Layer 3: Fused Linear + RELU *)
FOR j := 0 TO 11 DO
    sum := 0.0;
    FOR i := 0 TO 11 DO
        sum := sum + buffer_1[i] * weights_3[i * 12 + j];
    END_FOR;
buffer_0[j] := MAX(sum + bias_3[j], 0.0);
END_FOR;

(* Layer 4: Fused Linear + RELU *)
FOR j := 0 TO 11 DO
    sum := 0.0;
    FOR i := 0 TO 11 DO
        sum := sum + buffer_0[i] * weights_4[i * 12 + j];
    END_FOR;
buffer_1[j] := MAX(sum + bias_4[j], 0.0);
END_FOR;

(* Layer 5: Fused Linear + SOFTMAX *)
FOR j := 0 TO 2 DO
    sum := 0.0;
    FOR i := 0 TO 11 DO
        sum := sum + buffer_1[i] * weights_5[i * 3 + j];
    END_FOR;
output_data[j] := sum + bias_5[j];
END_FOR;

(* Softmax: find max *)
max_val := output_data[0];
FOR i := 1 TO 2 DO
    IF output_data[i] > max_val THEN
        max_val := output_data[i];
    END_IF;
END_FOR;

(* Softmax: compute exponentials and sum *)
exp_sum := 0.0;
FOR i := 0 TO 2 DO
    output_data[i] := EXP(output_data[i] - max_val);
    exp_sum := exp_sum + output_data[i];
END_FOR;

(* Softmax: normalize *)
FOR i := 0 TO 2 DO
    output_data[i] := output_data[i] / exp_sum;
END_FOR;

END_FUNCTION_BLOCK

(* ---- MLP5.st ---- *)
FUNCTION_BLOCK MLP5_FB

    (* Model Inputs/Outputs *)
VAR_INPUT
    input_data : REAL;
END_VAR

VAR_OUTPUT
    output_data : ARRAY[0..2] OF REAL;
END_VAR

VAR CONSTANT
    weights_0 : ARRAY[0..7] OF REAL := [-0.53507483, -0.669488788, -0.146161795, 0.430412263, 0.904008746, -0.046146214, -0.448489487, 0.180311218];
    bias_0 : ARRAY[0..7] OF REAL := [0, 0, 0, -0.0787891373, -0.0526719391, 0, 0, 0.0822643563];

    weights_1 : ARRAY[0..63] OF REAL := [0.063362658, 0.298499703, -0.57503885, -0.118522853, 0.0117590427, -0.340105176, 0.231563389, 0.172633767, -0.565162897, 0.377811849, -0.306341857, 0.105061293, 0.553966939, -0.387644529, 0.470730245, -0.538064957, -0.00107866526, 0.41243571, 0.100581408, -0.121569455, -0.492007643, 0.208534479, 0.00532305241, -0.477587283, 0.172095641, 0.0387620367, 0.382432431, 0.634039164, 0.780079305, 0.819513261, 0.754862785, -0.599698424, -0.400032878, 0.72033, 0.809848487, 0.425493389, 0.806156099, 0.838535607, 0.524595559, -0.600885093, -0.546205997, 0.0218340158, 0.546698272, -0.170108199, -0.593065739, -0.310147077, -0.0215710402, -0.520702839, 0.422134101, -0.229806542, -0.220874369, -0.386799335, -0.419301927, -0.0614820123, 0.192340791, 0.297955453, 0.237402886, 0.609429836, -0.0111329537, 0.207799405, 0.112620033, -0.307117581, -0.410346866, -0.0216449499];
    bias_1 : ARRAY[0..7] OF REAL := [0.0248198342, 0.127204463, -0.110540606, 0.0399958752, -0.0844260901, -0.0590777509, -0.0346453339, 0];

    weights_2 : ARRAY[0..63] OF REAL := [-0.288100004, -0.201139838, 1.06277561, 0.216839314, 0.188800827, -0.221569985, 0.222016305, 0.0345546268, -0.00159225659, -0.551148415, 0.769383252, 0.514585555, 0.443062097, 0.410166085, 0.270491093, 0.146244377, 0.67855072, -0.081202209, 0.194770858, 0.852390587, -0.581874967, 0.121784441, -0.205027789, 0.307291895, 0.00858160388, -0.0028219223, 0.456645638, 0.53842169, -0.0791837424, -0.334288418, 0.200156718, 0.14852111, 0.507059157, 0.131593883, 0.357866079, 0.197592288, -0.79305321, 0.264319122, 0.791967511, -0.604955614, 0.836388469, 0.465418398, -0.112717636, 0.0058227866, 0.165747017, 0.772809207, 0.563402057, -0.374170035, 0.752214313, -0.411610305, 0.00648151152, 0.0819479972, -0.525074184, -0.222901478, 0.738341391, -0.0950928926, 0.218107045, -0.335193545, -0.264200151, -0.522010565, -0.352673084, 0.462205946, 0.100470126, 0.130517006];
    bias_2 : ARRAY[0..7] OF REAL := [-0.0656886473, 0, 0.07456249, 0.0119883837, 0.124912612, -0.0470443293, -0.0403835066, -0.0663873032];

    weights_3 : ARRAY[0..63] OF REAL := [-0.406940758, -0.410205185, 0.841179371, 0.697039425, -0.796420038, 0.504597604, -0.270140171, -0.501359642, -0.0188109279, -0.174193621, 0.490450084, 0.205026269, -0.520047843, 0.569118798, -0.444546968, 0.163078547, -0.245197535, -0.00735265808, 0.753572881, 0.32959187, 0.250873566, 0.624375761, -0.34793222, 0.638749421, 0.287776947, 0.304210067, 0.540278256, 0.592640877, 0.117994718, 0.22743687, -0.525758684, -0.55700624, -0.394151956, -0.321884453, -0.141238824, -0.726398766, 0.542078376, -0.403606266, 0.359072655, 0.831410825, 0.0812664628, 0.0501168296, -0.350325465, 0.337302566, 0.176324472, 0.707275867, 0.257912636, -0.325850964, -0.144438624, -0.561803877, 0.295645416, 0.369945198, -0.211105391, 0.857302606, 0.464602023, 0.400751472, -0.427103639, 0.531412184, -0.571155608, 0.32104066, 0.168936327, 0.228739277, -0.341044396, -0.495310009];
    bias_3 : ARRAY[0..7] OF REAL := [0, -0.0137715843, 0.094763279, -0.0867965817, 0.12138544, -0.0279933698, -0.0032245568, 0.14148654];

    weights_4 : ARRAY[0..63] OF REAL := [-0.369385809, 0.435406744, 0.0232670307, -0.334486037, -0.180559844, 0.432826102, -0.18959716, -0.286127001, 0.159696162, 0.0740950704, 0.190330386, -0.362739533, 0.370848238, 0.303789914, 0.440430582, 0.302749634, -0.595516324, -0.123227149, 0.276114434, 0.178365439, 0.459796816, -0.0895816684, 0.450091243, 0.504246593, -0.347878426, -0.421078503, -0.0440155193, 0.405472338, 0.693396926, -0.301305711, -0.378517181, 0.438089758, 0.138437688, -0.250610679, -0.414459199, -0.664958417, 0.293263495, -0.123279721, 0.470128387, -0.754871607, -0.333532512, -0.284029275, -0.303617388, 0.800206959, 0.418326527, -0.518932998, 0.306997985, 0.203854516, -0.441367209, 0.0111179948, -0.552968621, 0.449602693, -0.512903392, 0.0850611925, -0.399994045, -0.0910809636, -0.104376674, -0.196162522, 0.0364336371, -0.0938068181, 0.0166178457, -0.528001726, 0.6952039, 0.0915063098];
    bias_4 : ARRAY[0..7] OF REAL := [0, 0, -0.0477878414, -0.0651340261, 0.184870526, 0, 0.227151066, -0.0231719129];

    weights_5 : ARRAY[0..63] OF REAL := [0.0587205887, 0.0533784032, 0.158940315, -0.107622564, -0.145722538, -0.00944948196, 0.529260933, 0.0305299759, -0.174156368, 0.400077522, -0.36074695, 0.0345277786, -0.473972589, 0.147112012, -0.429324031, -0.177337885, 0.32189554, -0.154660687, -0.606729031, 0.123603523, -0.170367599, -0.502868116, -0.0876729265, 0.114311762, 0.707142949, -0.366575629, 0.0513379686, -0.494380474, -0.826889455, 0.679591119, 0.792746127, -0.579329967, 0.683867276, 0.297326177, -0.0109938271, 0.135385692, 0.176608101, 0.521379054, -0.266024411, 0.23239027, 0.0833909512, -0.428257197, 0.17536968, -0.310296744, 0.470981777, -0.0650536418, -0.242025822, 0.180521727, -0.209767953, 0.0444659442, 0.625916123, -0.291563928, 0.629532635, 0.446459383, 0.29174152, 0.729171097, 0.344551712, -0.182016864, 0.39470911, -0.429122269, 0.202520087, 0.931188405, 0.796285152, -0.478577644];
    bias_5 : ARRAY[0..7] OF REAL := [-0.0112341903, 0.107019141, 0.194828868, 0, 0.0908448994, 0.0031164973, 0.0566227362, 0.183672369];

    weights_6 : ARRAY[0..63] OF REAL := [-0.500871062, -0.0426991582, -0.325405121, 0.0876715183, 0.627584994, -0.135081053, -0.556043506, -0.608783484, -0.258675456, 0.0234838128, -0.0112303877, -0.233016968, -0.435161024, 0.115634076, -0.299919873, -0.414022267, 0.372731984, -0.56812948, -0.0739866197, 0.24208802, 0.0946503058, 0.154511169, 0.0714637041, 0.174022198, 0.500243008, 0.324402034, -0.165571511, 0.101269364, 0.555786908, 0.0490795374, -0.10130465, -0.404081643, 0.334687829, 0.205921113, 0.148157805, -0.610701621, -0.43316859, 0.658870935, 0.127036929, -0.435543954, -0.610272408, -0.387020975, -0.453532517, -0.502265394, 0.781038046, -0.0541303866, -0.589179754, -0.249233156, -0.259051144, -0.0262311101, 0.451682925, -0.0268176198, 0.659966707, 0.160063073, -0.345124543, 0.46368593, -0.0950434208, -0.23101297, 0.208650693, -0.120401442, -0.740491629, 0.86507839, -0.583369792, 0.498632133];
    bias_6 : ARRAY[0..7] OF REAL := [0, 0, -0.0134519087, 0, 0.0197975468, 0.238473833, 0, 0];

    weights_7 : ARRAY[0..63] OF REAL := [0.0472229719, 0.499810636, -0.323982716, 0.11469543, -0.375817299, 0.219568372, -0.263723314, -0.434796005, 0.471136868, -0.0162989497, -0.428802371, 0.53169769, 0.471080363, 0.11451906, -0.33936584, 0.241111815, -0.475392103, -0.0629273057, -0.593522727, -0.430725843, -0.416154951, -0.104646206, -0.577033043, -0.295274824, -0.0381647944, -0.22522971, -0.457870573, 0.0317639709, -0.242461175, -0.581591249, 0.30567652, 0.155042946, 0.644507229, 0.736880124, -0.142929405, -0.658658862, 0.766304135, -0.430037975, 0.00776856299, 0.572000384, 0.0853363872, -0.450751841, -0.328342885, 0.525618732, 0.114655629, -0.388185203, -0.251179636, 0.835268259, 0.603164017, -0.0067243576, 0.219419897, -0.324196905, 0.368480742, 0.111086726, -0.0390381813, -0.0325580835, -0.306076735, -0.0825812221, -0.211727262, 0.14168328, -0.268856406, 0.353065252, 0.103686988, 0.4429757];
    bias_7 : ARRAY[0..7] OF REAL := [-0.205431893, -0.0555614866, 0, 0.144488201, -0.1497363, 0, -0.0637752041, 0.459758997];

    weights_8 : ARRAY[0..63] OF REAL := [-0.197457016, 0.141665965, -0.359861732, -0.132918373, -0.342840284, 0.475130945, 0.429878056, 0.057383772, -0.0928481221, -0.370261163, -0.392136157, -0.258805513, -0.0142944586, 0.322692961, -0.344118297, 0.735266209, -0.448836923, -0.544512093, 0.307438493, -0.373555899, 0.574374378, 0.475989759, 0.237792373, 0.565786898, 0.715095699, 0.942202628, 0.188565761, 0.890218079, 0.996486366, -0.837896883, -0.0032916069, 0.691578329, 0.302878022, -0.442298859, 0.424598515, -0.254163921, 0.148600698, 0.644482732, 0.02359128, 0.35823977, -0.230832934, -0.329942495, -0.446255922, -0.0825818181, -0.111995578, 0.0555180311, -0.210629761, -0.551132798, -0.449758619, -0.425730079, 0.366501093, 0.330503494, 0.571831942, -0.330727249, -0.243855655, 0.0638255477, -0.113650091, 0.637051284, 0.715611696, 0.803717911, 0.0760587007, 0.521238744, -0.491941065, 0.801276624];
    bias_8 : ARRAY[0..7] OF REAL := [0.0661619008, 0.211298704, 0.352757961, 0.31050095, 0.290936738, -0.136591047, 0, 0.342236161];

    weights_9 : ARRAY[0..63] OF REAL := [-0.52104789, 0.460638374, 0.0360075086, -0.00834363699, 0.483171791, 0.304018676, -0.10147053, -0.531910062, -0.90199554, -0.0968902409, 1.02613008, -0.305097938, 0.247813627, -0.382043809, -0.146120548, -0.794718981, 0.363161296, 0.450564861, 0.406178683, -0.227152258, 0.782353103, -0.158298492, -0.357196778, 0.239361629, 0.275576204, 0.734804451, 1.00428867, 0.41201967, 0.826547801, 0.294418097, -0.0447072387, -0.306748569, 0.197246879, 0.588557303, 0.778613269, 0.141008914, 0.328565836, 0.489948213, -0.318891525, -0.601634741, 0.813271165, -0.391228199, -0.301011592, -0.412705481, -0.336696744, -0.153892338, -0.370729327, 0.883742392, -0.499530792, -0.171516687, 0.570708215, 0.537043393, 0.529110491, 0.101749957, -0.116467595, -0.527576983, 0.307871729, 0.411601573, 0.599725902, -0.328691691, -0.00560221449, -0.326922148, -0.159318447, 0.475381225];
    bias_9 : ARRAY[0..7] OF REAL := [-0.0623566136, 0.197932214, 0.296277493, 0, 0.250260174, 0, 0, 0.0349539854];

    weights_10 : ARRAY[0..63] OF REAL := [-0.163975596, -0.239289299, 0.838056445, -0.0944938883, 0.3310121, 0.0772968307, -0.125489324, 0.601332784, -0.129733533, -0.479307264, -0.266973853, 0.274074376, -0.168107465, 0.837115288, 0.808397591, -0.415453404, -0.543875217, 0.0343489945, 0.305932015, -0.565567851, 0.883265436, 0.72432363, 0.646220267, -0.482283801, 0.302705884, -0.555842519, 0.086917758, 0.337820709, 0.270993114, 0.177294791, -0.242245823, 0.502743304, 0.027063787, 0.412451118, -0.229175135, -1.04114318, 0.676691353, -0.0671654865, 0.847393811, -0.6518296, 0.560024083, 0.334516823, -0.0695735216, -0.358827323, -0.353390962, -0.0454823971, 0.462751925, -0.015168786, -0.260765046, -0.0559414625, -0.331326127, -0.0680848956, 0.409886062, -0.266761303, 0.251534104, -0.588591099, -0.324441016, -0.138969421, 1.03054678, 0.731393456, -0.731957138, -0.339184999, -0.0591701046, 0.112207964];
    bias_10 : ARRAY[0..7] OF REAL := [0, -0.104845211, -0.0487807542, -0.253034264, 0.176031917, 0.276837677, 0.317505389, -0.224763602];

    weights_11 : ARRAY[0..23] OF REAL := [-0.356673032, -0.18541801, 0.28275007, -0.566354752, -0.0957784876, -0.813595474, -1.27709067, 0.593999088, 0.798196673, -0.309898615, -0.546126246, 0.484500587, 0.201039955, -0.676716924, -1.46589875, 0.101248577, 0.0413070917, -0.947486281, 0.722890437, 0.790142775, -0.549232304, 0.500470102, -0.795395613, 0.884318352];
    bias_11 : ARRAY[0..2] OF REAL := [0.0316488892, 0.198421121, -0.224571243];

END_VAR

VAR
    (* Merged variables from all regions *)
    buffer_0 : ARRAY[0..7] OF REAL;
    buffer_1 : ARRAY[0..7] OF REAL;

    (* Temporary computation variables *)
    i : DINT;
    j : DINT;
    t : DINT;
    sum : REAL;
    (* Computation helpers *)
    max_val : REAL;
    exp_val : REAL;
    exp_sum : REAL;
    (* Spatial loop variables *)
    oc : DINT;
    oh : DINT;
    ow : DINT;
    ic : DINT;
    kh : DINT;
    kw : DINT;
    ih : DINT;
    iw : DINT;
END_VAR

(* Forward pass execution *)

(* Region: r0 [ACYCLIC] *)
(* Acyclic Region r0 *)
(* Layer 0: Fused Linear + RELU *)
FOR j := 0 TO 7 DO
    sum := 0.0;
    FOR i := 0 TO 0 DO
        sum := sum + input_data * weights_0[i * 8 + j];
    END_FOR;
buffer_1[j] := MAX(sum + bias_0[j], 0.0);
END_FOR;

(* Layer 1: Fused Linear + RELU *)
FOR j := 0 TO 7 DO
    sum := 0.0;
    FOR i := 0 TO 7 DO
        sum := sum + buffer_1[i] * weights_1[i * 8 + j];
    END_FOR;
buffer_0[j] := MAX(sum + bias_1[j], 0.0);
END_FOR;

(* Layer 2: Fused Linear + RELU *)
FOR j := 0 TO 7 DO
    sum := 0.0;
    FOR i := 0 TO 7 DO
        sum := sum + buffer_0[i] * weights_2[i * 8 + j];
    END_FOR;
buffer_1[j] := MAX(sum + bias_2[j], 0.0);
END_FOR;

(* Layer 3: Fused Linear + RELU *)
FOR j := 0 TO 7 DO
    sum := 0.0;
    FOR i := 0 TO 7 DO
        sum := sum + buffer_1[i] * weights_3[i * 8 + j];
    END_FOR;
buffer_0[j] := MAX(sum + bias_3[j], 0.0);
END_FOR;

(* Layer 4: Fused Linear + RELU *)
FOR j := 0 TO 7 DO
    sum := 0.0;
    FOR i := 0 TO 7 DO
        sum := sum + buffer_0[i] * weights_4[i * 8 + j];
    END_FOR;
buffer_1[j] := MAX(sum + bias_4[j], 0.0);
END_FOR;

(* Layer 5: Fused Linear + RELU *)
FOR j := 0 TO 7 DO
    sum := 0.0;
    FOR i := 0 TO 7 DO
        sum := sum + buffer_1[i] * weights_5[i * 8 + j];
    END_FOR;
buffer_0[j] := MAX(sum + bias_5[j], 0.0);
END_FOR;

(* Layer 6: Fused Linear + RELU *)
FOR j := 0 TO 7 DO
    sum := 0.0;
    FOR i := 0 TO 7 DO
        sum := sum + buffer_0[i] * weights_6[i * 8 + j];
    END_FOR;
buffer_1[j] := MAX(sum + bias_6[j], 0.0);
END_FOR;

(* Layer 7: Fused Linear + RELU *)
FOR j := 0 TO 7 DO
    sum := 0.0;
    FOR i := 0 TO 7 DO
        sum := sum + buffer_1[i] * weights_7[i * 8 + j];
    END_FOR;
buffer_0[j] := MAX(sum + bias_7[j], 0.0);
END_FOR;

(* Layer 8: Fused Linear + RELU *)
FOR j := 0 TO 7 DO
    sum := 0.0;
    FOR i := 0 TO 7 DO
        sum := sum + buffer_0[i] * weights_8[i * 8 + j];
    END_FOR;
buffer_1[j] := MAX(sum + bias_8[j], 0.0);
END_FOR;

(* Layer 9: Fused Linear + RELU *)
FOR j := 0 TO 7 DO
    sum := 0.0;
    FOR i := 0 TO 7 DO
        sum := sum + buffer_1[i] * weights_9[i * 8 + j];
    END_FOR;
buffer_0[j] := MAX(sum + bias_9[j], 0.0);
END_FOR;

(* Layer 10: Fused Linear + RELU *)
FOR j := 0 TO 7 DO
    sum := 0.0;
    FOR i := 0 TO 7 DO
        sum := sum + buffer_0[i] * weights_10[i * 8 + j];
    END_FOR;
buffer_1[j] := MAX(sum + bias_10[j], 0.0);
END_FOR;

(* Layer 11: Fused Linear + SOFTMAX *)
FOR j := 0 TO 2 DO
    sum := 0.0;
    FOR i := 0 TO 7 DO
        sum := sum + buffer_1[i] * weights_11[i * 3 + j];
    END_FOR;
output_data[j] := sum + bias_11[j];
END_FOR;

(* Softmax: find max *)
max_val := output_data[0];
FOR i := 1 TO 2 DO
    IF output_data[i] > max_val THEN
        max_val := output_data[i];
    END_IF;
END_FOR;

(* Softmax: compute exponentials and sum *)
exp_sum := 0.0;
FOR i := 0 TO 2 DO
    output_data[i] := EXP(output_data[i] - max_val);
    exp_sum := exp_sum + output_data[i];
END_FOR;

(* Softmax: normalize *)
FOR i := 0 TO 2 DO
    output_data[i] := output_data[i] / exp_sum;
END_FOR;

END_FUNCTION_BLOCK

(* ---- MLP5_straton.st ---- *)
FUNCTION_BLOCK MLP5_FB

    (* Model Inputs/Outputs *)
VAR_INPUT
    input_data : REAL;
END_VAR

VAR_OUTPUT
    output_data : ARRAY[0..2] OF REAL;
END_VAR

VAR
    CONSTANT weights_0 : ARRAY[0..7] OF REAL := [-0.53507483, -0.669488788, -0.146161795, 0.430412263, 0.904008746, -0.046146214, -0.448489487, 0.180311218];
    CONSTANT bias_0 : ARRAY[0..7] OF REAL := [0, 0, 0, -0.0787891373, -0.0526719391, 0, 0, 0.0822643563];
    CONSTANT weights_1 : ARRAY[0..63] OF REAL := [0.063362658, 0.298499703, -0.57503885, -0.118522853, 0.0117590427, -0.340105176, 0.231563389, 0.172633767, -0.565162897, 0.377811849, -0.306341857, 0.105061293, 0.553966939, -0.387644529, 0.470730245, -0.538064957, -0.00107866526, 0.41243571, 0.100581408, -0.121569455, -0.492007643, 0.208534479, 0.00532305241, -0.477587283, 0.172095641, 0.0387620367, 0.382432431, 0.634039164, 0.780079305, 0.819513261, 0.754862785, -0.599698424, -0.400032878, 0.72033, 0.809848487, 0.425493389, 0.806156099, 0.838535607, 0.524595559, -0.600885093, -0.546205997, 0.0218340158, 0.546698272, -0.170108199, -0.593065739, -0.310147077, -0.0215710402, -0.520702839, 0.422134101, -0.229806542, -0.220874369, -0.386799335, -0.419301927, -0.0614820123, 0.192340791, 0.297955453, 0.237402886, 0.609429836, -0.0111329537, 0.207799405, 0.112620033, -0.307117581, -0.410346866, -0.0216449499];
    CONSTANT bias_1 : ARRAY[0..7] OF REAL := [0.0248198342, 0.127204463, -0.110540606, 0.0399958752, -0.0844260901, -0.0590777509, -0.0346453339, 0];
    CONSTANT weights_2 : ARRAY[0..63] OF REAL := [-0.288100004, -0.201139838, 1.06277561, 0.216839314, 0.188800827, -0.221569985, 0.222016305, 0.0345546268, -0.00159225659, -0.551148415, 0.769383252, 0.514585555, 0.443062097, 0.410166085, 0.270491093, 0.146244377, 0.67855072, -0.081202209, 0.194770858, 0.852390587, -0.581874967, 0.121784441, -0.205027789, 0.307291895, 0.00858160388, -0.0028219223, 0.456645638, 0.53842169, -0.0791837424, -0.334288418, 0.200156718, 0.14852111, 0.507059157, 0.131593883, 0.357866079, 0.197592288, -0.79305321, 0.264319122, 0.791967511, -0.604955614, 0.836388469, 0.465418398, -0.112717636, 0.0058227866, 0.165747017, 0.772809207, 0.563402057, -0.374170035, 0.752214313, -0.411610305, 0.00648151152, 0.0819479972, -0.525074184, -0.222901478, 0.738341391, -0.0950928926, 0.218107045, -0.335193545, -0.264200151, -0.522010565, -0.352673084, 0.462205946, 0.100470126, 0.130517006];
    CONSTANT bias_2 : ARRAY[0..7] OF REAL := [-0.0656886473, 0, 0.07456249, 0.0119883837, 0.124912612, -0.0470443293, -0.0403835066, -0.0663873032];
    CONSTANT weights_3 : ARRAY[0..63] OF REAL := [-0.406940758, -0.410205185, 0.841179371, 0.697039425, -0.796420038, 0.504597604, -0.270140171, -0.501359642, -0.0188109279, -0.174193621, 0.490450084, 0.205026269, -0.520047843, 0.569118798, -0.444546968, 0.163078547, -0.245197535, -0.00735265808, 0.753572881, 0.32959187, 0.250873566, 0.624375761, -0.34793222, 0.638749421, 0.287776947, 0.304210067, 0.540278256, 0.592640877, 0.117994718, 0.22743687, -0.525758684, -0.55700624, -0.394151956, -0.321884453, -0.141238824, -0.726398766, 0.542078376, -0.403606266, 0.359072655, 0.831410825, 0.0812664628, 0.0501168296, -0.350325465, 0.337302566, 0.176324472, 0.707275867, 0.257912636, -0.325850964, -0.144438624, -0.561803877, 0.295645416, 0.369945198, -0.211105391, 0.857302606, 0.464602023, 0.400751472, -0.427103639, 0.531412184, -0.571155608, 0.32104066, 0.168936327, 0.228739277, -0.341044396, -0.495310009];
    CONSTANT bias_3 : ARRAY[0..7] OF REAL := [0, -0.0137715843, 0.094763279, -0.0867965817, 0.12138544, -0.0279933698, -0.0032245568, 0.14148654];
    CONSTANT weights_4 : ARRAY[0..63] OF REAL := [-0.369385809, 0.435406744, 0.0232670307, -0.334486037, -0.180559844, 0.432826102, -0.18959716, -0.286127001, 0.159696162, 0.0740950704, 0.190330386, -0.362739533, 0.370848238, 0.303789914, 0.440430582, 0.302749634, -0.595516324, -0.123227149, 0.276114434, 0.178365439, 0.459796816, -0.0895816684, 0.450091243, 0.504246593, -0.347878426, -0.421078503, -0.0440155193, 0.405472338, 0.693396926, -0.301305711, -0.378517181, 0.438089758, 0.138437688, -0.250610679, -0.414459199, -0.664958417, 0.293263495, -0.123279721, 0.470128387, -0.754871607, -0.333532512, -0.284029275, -0.303617388, 0.800206959, 0.418326527, -0.518932998, 0.306997985, 0.203854516, -0.441367209, 0.0111179948, -0.552968621, 0.449602693, -0.512903392, 0.0850611925, -0.399994045, -0.0910809636, -0.104376674, -0.196162522, 0.0364336371, -0.0938068181, 0.0166178457, -0.528001726, 0.6952039, 0.0915063098];
    CONSTANT bias_4 : ARRAY[0..7] OF REAL := [0, 0, -0.0477878414, -0.0651340261, 0.184870526, 0, 0.227151066, -0.0231719129];
    CONSTANT weights_5 : ARRAY[0..63] OF REAL := [0.0587205887, 0.0533784032, 0.158940315, -0.107622564, -0.145722538, -0.00944948196, 0.529260933, 0.0305299759, -0.174156368, 0.400077522, -0.36074695, 0.0345277786, -0.473972589, 0.147112012, -0.429324031, -0.177337885, 0.32189554, -0.154660687, -0.606729031, 0.123603523, -0.170367599, -0.502868116, -0.0876729265, 0.114311762, 0.707142949, -0.366575629, 0.0513379686, -0.494380474, -0.826889455, 0.679591119, 0.792746127, -0.579329967, 0.683867276, 0.297326177, -0.0109938271, 0.135385692, 0.176608101, 0.521379054, -0.266024411, 0.23239027, 0.0833909512, -0.428257197, 0.17536968, -0.310296744, 0.470981777, -0.0650536418, -0.242025822, 0.180521727, -0.209767953, 0.0444659442, 0.625916123, -0.291563928, 0.629532635, 0.446459383, 0.29174152, 0.729171097, 0.344551712, -0.182016864, 0.39470911, -0.429122269, 0.202520087, 0.931188405, 0.796285152, -0.478577644];
    CONSTANT bias_5 : ARRAY[0..7] OF REAL := [-0.0112341903, 0.107019141, 0.194828868, 0, 0.0908448994, 0.0031164973, 0.0566227362, 0.183672369];
    CONSTANT weights_6 : ARRAY[0..63] OF REAL := [-0.500871062, -0.0426991582, -0.325405121, 0.0876715183, 0.627584994, -0.135081053, -0.556043506, -0.608783484, -0.258675456, 0.0234838128, -0.0112303877, -0.233016968, -0.435161024, 0.115634076, -0.299919873, -0.414022267, 0.372731984, -0.56812948, -0.0739866197, 0.24208802, 0.0946503058, 0.154511169, 0.0714637041, 0.174022198, 0.500243008, 0.324402034, -0.165571511, 0.101269364, 0.555786908, 0.0490795374, -0.10130465, -0.404081643, 0.334687829, 0.205921113, 0.148157805, -0.610701621, -0.43316859, 0.658870935, 0.127036929, -0.435543954, -0.610272408, -0.387020975, -0.453532517, -0.502265394, 0.781038046, -0.0541303866, -0.589179754, -0.249233156, -0.259051144, -0.0262311101, 0.451682925, -0.0268176198, 0.659966707, 0.160063073, -0.345124543, 0.46368593, -0.0950434208, -0.23101297, 0.208650693, -0.120401442, -0.740491629, 0.86507839, -0.583369792, 0.498632133];
    CONSTANT bias_6 : ARRAY[0..7] OF REAL := [0, 0, -0.0134519087, 0, 0.0197975468, 0.238473833, 0, 0];
    CONSTANT weights_7 : ARRAY[0..63] OF REAL := [0.0472229719, 0.499810636, -0.323982716, 0.11469543, -0.375817299, 0.219568372, -0.263723314, -0.434796005, 0.471136868, -0.0162989497, -0.428802371, 0.53169769, 0.471080363, 0.11451906, -0.33936584, 0.241111815, -0.475392103, -0.0629273057, -0.593522727, -0.430725843, -0.416154951, -0.104646206, -0.577033043, -0.295274824, -0.0381647944, -0.22522971, -0.457870573, 0.0317639709, -0.242461175, -0.581591249, 0.30567652, 0.155042946, 0.644507229, 0.736880124, -0.142929405, -0.658658862, 0.766304135, -0.430037975, 0.00776856299, 0.572000384, 0.0853363872, -0.450751841, -0.328342885, 0.525618732, 0.114655629, -0.388185203, -0.251179636, 0.835268259, 0.603164017, -0.0067243576, 0.219419897, -0.324196905, 0.368480742, 0.111086726, -0.0390381813, -0.0325580835, -0.306076735, -0.0825812221, -0.211727262, 0.14168328, -0.268856406, 0.353065252, 0.103686988, 0.4429757];
    CONSTANT bias_7 : ARRAY[0..7] OF REAL := [-0.205431893, -0.0555614866, 0, 0.144488201, -0.1497363, 0, -0.0637752041, 0.459758997];
    CONSTANT weights_8 : ARRAY[0..63] OF REAL := [-0.197457016, 0.141665965, -0.359861732, -0.132918373, -0.342840284, 0.475130945, 0.429878056, 0.057383772, -0.0928481221, -0.370261163, -0.392136157, -0.258805513, -0.0142944586, 0.322692961, -0.344118297, 0.735266209, -0.448836923, -0.544512093, 0.307438493, -0.373555899, 0.574374378, 0.475989759, 0.237792373, 0.565786898, 0.715095699, 0.942202628, 0.188565761, 0.890218079, 0.996486366, -0.837896883, -0.0032916069, 0.691578329, 0.302878022, -0.442298859, 0.424598515, -0.254163921, 0.148600698, 0.644482732, 0.02359128, 0.35823977, -0.230832934, -0.329942495, -0.446255922, -0.0825818181, -0.111995578, 0.0555180311, -0.210629761, -0.551132798, -0.449758619, -0.425730079, 0.366501093, 0.330503494, 0.571831942, -0.330727249, -0.243855655, 0.0638255477, -0.113650091, 0.637051284, 0.715611696, 0.803717911, 0.0760587007, 0.521238744, -0.491941065, 0.801276624];
    CONSTANT bias_8 : ARRAY[0..7] OF REAL := [0.0661619008, 0.211298704, 0.352757961, 0.31050095, 0.290936738, -0.136591047, 0, 0.342236161];
    CONSTANT weights_9 : ARRAY[0..63] OF REAL := [-0.52104789, 0.460638374, 0.0360075086, -0.00834363699, 0.483171791, 0.304018676, -0.10147053, -0.531910062, -0.90199554, -0.0968902409, 1.02613008, -0.305097938, 0.247813627, -0.382043809, -0.146120548, -0.794718981, 0.363161296, 0.450564861, 0.406178683, -0.227152258, 0.782353103, -0.158298492, -0.357196778, 0.239361629, 0.275576204, 0.734804451, 1.00428867, 0.41201967, 0.826547801, 0.294418097, -0.0447072387, -0.306748569, 0.197246879, 0.588557303, 0.778613269, 0.141008914, 0.328565836, 0.489948213, -0.318891525, -0.601634741, 0.813271165, -0.391228199, -0.301011592, -0.412705481, -0.336696744, -0.153892338, -0.370729327, 0.883742392, -0.499530792, -0.171516687, 0.570708215, 0.537043393, 0.529110491, 0.101749957, -0.116467595, -0.527576983, 0.307871729, 0.411601573, 0.599725902, -0.328691691, -0.00560221449, -0.326922148, -0.159318447, 0.475381225];
    CONSTANT bias_9 : ARRAY[0..7] OF REAL := [-0.0623566136, 0.197932214, 0.296277493, 0, 0.250260174, 0, 0, 0.0349539854];
    CONSTANT weights_10 : ARRAY[0..63] OF REAL := [-0.163975596, -0.239289299, 0.838056445, -0.0944938883, 0.3310121, 0.0772968307, -0.125489324, 0.601332784, -0.129733533, -0.479307264, -0.266973853, 0.274074376, -0.168107465, 0.837115288, 0.808397591, -0.415453404, -0.543875217, 0.0343489945, 0.305932015, -0.565567851, 0.883265436, 0.72432363, 0.646220267, -0.482283801, 0.302705884, -0.555842519, 0.086917758, 0.337820709, 0.270993114, 0.177294791, -0.242245823, 0.502743304, 0.027063787, 0.412451118, -0.229175135, -1.04114318, 0.676691353, -0.0671654865, 0.847393811, -0.6518296, 0.560024083, 0.334516823, -0.0695735216, -0.358827323, -0.353390962, -0.0454823971, 0.462751925, -0.015168786, -0.260765046, -0.0559414625, -0.331326127, -0.0680848956, 0.409886062, -0.266761303, 0.251534104, -0.588591099, -0.324441016, -0.138969421, 1.03054678, 0.731393456, -0.731957138, -0.339184999, -0.0591701046, 0.112207964];
    CONSTANT bias_10 : ARRAY[0..7] OF REAL := [0, -0.104845211, -0.0487807542, -0.253034264, 0.176031917, 0.276837677, 0.317505389, -0.224763602];
    CONSTANT weights_11 : ARRAY[0..23] OF REAL := [-0.356673032, -0.18541801, 0.28275007, -0.566354752, -0.0957784876, -0.813595474, -1.27709067, 0.593999088, 0.798196673, -0.309898615, -0.546126246, 0.484500587, 0.201039955, -0.676716924, -1.46589875, 0.101248577, 0.0413070917, -0.947486281, 0.722890437, 0.790142775, -0.549232304, 0.500470102, -0.795395613, 0.884318352];
    CONSTANT bias_11 : ARRAY[0..2] OF REAL := [0.0316488892, 0.198421121, -0.224571243];
END_VAR

VAR
    (* Merged variables from all regions *)
    buffer_0 : ARRAY[0..7] OF REAL;
    buffer_1 : ARRAY[0..7] OF REAL;

    (* Temporary computation variables *)
    i : DINT;
    j : DINT;
    t : DINT;
    sum : REAL;
    (* Computation helpers *)
    max_val : REAL;
    exp_val : REAL;
    exp_sum : REAL;
    (* Spatial loop variables *)
    oc : DINT;
    oh : DINT;
    ow : DINT;
    ic : DINT;
    kh : DINT;
    kw : DINT;
    ih : DINT;
    iw : DINT;
END_VAR

(* Forward pass execution *)

(* Region: r0 [ACYCLIC] *)
(* Acyclic Region r0 *)
(* Layer 0: Fused Linear + RELU *)
FOR j := 0 TO 7 DO
    sum := 0.0;
    FOR i := 0 TO 0 DO
        sum := sum + input_data * weights_0[i * 8 + j];
    END_FOR;
buffer_1[j] := MAX(sum + bias_0[j], 0.0);
END_FOR;

(* Layer 1: Fused Linear + RELU *)
FOR j := 0 TO 7 DO
    sum := 0.0;
    FOR i := 0 TO 7 DO
        sum := sum + buffer_1[i] * weights_1[i * 8 + j];
    END_FOR;
buffer_0[j] := MAX(sum + bias_1[j], 0.0);
END_FOR;

(* Layer 2: Fused Linear + RELU *)
FOR j := 0 TO 7 DO
    sum := 0.0;
    FOR i := 0 TO 7 DO
        sum := sum + buffer_0[i] * weights_2[i * 8 + j];
    END_FOR;
buffer_1[j] := MAX(sum + bias_2[j], 0.0);
END_FOR;

(* Layer 3: Fused Linear + RELU *)
FOR j := 0 TO 7 DO
    sum := 0.0;
    FOR i := 0 TO 7 DO
        sum := sum + buffer_1[i] * weights_3[i * 8 + j];
    END_FOR;
buffer_0[j] := MAX(sum + bias_3[j], 0.0);
END_FOR;

(* Layer 4: Fused Linear + RELU *)
FOR j := 0 TO 7 DO
    sum := 0.0;
    FOR i := 0 TO 7 DO
        sum := sum + buffer_0[i] * weights_4[i * 8 + j];
    END_FOR;
buffer_1[j] := MAX(sum + bias_4[j], 0.0);
END_FOR;

(* Layer 5: Fused Linear + RELU *)
FOR j := 0 TO 7 DO
    sum := 0.0;
    FOR i := 0 TO 7 DO
        sum := sum + buffer_1[i] * weights_5[i * 8 + j];
    END_FOR;
buffer_0[j] := MAX(sum + bias_5[j], 0.0);
END_FOR;

(* Layer 6: Fused Linear + RELU *)
FOR j := 0 TO 7 DO
    sum := 0.0;
    FOR i := 0 TO 7 DO
        sum := sum + buffer_0[i] * weights_6[i * 8 + j];
    END_FOR;
buffer_1[j] := MAX(sum + bias_6[j], 0.0);
END_FOR;

(* Layer 7: Fused Linear + RELU *)
FOR j := 0 TO 7 DO
    sum := 0.0;
    FOR i := 0 TO 7 DO
        sum := sum + buffer_1[i] * weights_7[i * 8 + j];
    END_FOR;
buffer_0[j] := MAX(sum + bias_7[j], 0.0);
END_FOR;

(* Layer 8: Fused Linear + RELU *)
FOR j := 0 TO 7 DO
    sum := 0.0;
    FOR i := 0 TO 7 DO
        sum := sum + buffer_0[i] * weights_8[i * 8 + j];
    END_FOR;
buffer_1[j] := MAX(sum + bias_8[j], 0.0);
END_FOR;

(* Layer 9: Fused Linear + RELU *)
FOR j := 0 TO 7 DO
    sum := 0.0;
    FOR i := 0 TO 7 DO
        sum := sum + buffer_1[i] * weights_9[i * 8 + j];
    END_FOR;
buffer_0[j] := MAX(sum + bias_9[j], 0.0);
END_FOR;

(* Layer 10: Fused Linear + RELU *)
FOR j := 0 TO 7 DO
    sum := 0.0;
    FOR i := 0 TO 7 DO
        sum := sum + buffer_0[i] * weights_10[i * 8 + j];
    END_FOR;
buffer_1[j] := MAX(sum + bias_10[j], 0.0);
END_FOR;

(* Layer 11: Fused Linear + SOFTMAX *)
FOR j := 0 TO 2 DO
    sum := 0.0;
    FOR i := 0 TO 7 DO
        sum := sum + buffer_1[i] * weights_11[i * 3 + j];
    END_FOR;
output_data[j] := sum + bias_11[j];
END_FOR;

(* Softmax: find max *)
max_val := output_data[0];
FOR i := 1 TO 2 DO
    IF output_data[i] > max_val THEN
        max_val := output_data[i];
    END_IF;
END_FOR;

(* Softmax: compute exponentials and sum *)
exp_sum := 0.0;
FOR i := 0 TO 2 DO
    output_data[i] := EXP(output_data[i] - max_val);
    exp_sum := exp_sum + output_data[i];
END_FOR;

(* Softmax: normalize *)
FOR i := 0 TO 2 DO
    output_data[i] := output_data[i] / exp_sum;
END_FOR;

END_FUNCTION_BLOCK
